(* Scaling ******************************************************************)
	IF MaxValue <> MinValue 
	THEN
		Q 													:= Offset + Scale(In , SEL(Options.0, 0.0, SEL(Options.4, -32768.0, -7629.0)), 32767.0, MinValue , MaxValue);
		IF NoOfDigits > 0
		THEN
			Q												:= TO_FMLREAL(Q,NoOfDigits);
		END_IF
	
	ELSIF NoOfDigits > 0 (* Bsp PT100 *)
	THEN
		Q													:= Offset + TO_FMLREAL(In,NoOfDigits);
		
	ELSE  													
		Q 													:= 0.0;
	END_IF

	IF 	Error AND OutOnError <> 0.000000000000000001
	THEN
		Q													:= OutOnError;
	END_IF
(**********************************************************************************************************************)

{attribute 'monitoring' := 'call'}
PROPERTY PUBLIC Error : BOOL
GET
Error					:= Status.6 OR MinValue = MaxValue AND NoOfDigits = 0;
END_GET
END_PROPERTY

{attribute 'monitoring' := 'call'}
PROPERTY PUBLIC Limit_1 : BYTE
GET
Limit_1.0					:= Status.2;
Limit_1.1					:= Status.3;
END_GET
END_PROPERTY

{attribute 'monitoring' := 'call'}
PROPERTY PUBLIC Limit_2 : BYTE
GET
Limit_2.0					:= Status.4;
Limit_2.1					:= Status.5;
END_GET
END_PROPERTY

PROPERTY PUBLIC optEnableScaleExtRangeModeNeg7629 : bool
GET
optEnableScaleExtRangeModeNeg7629 := Options.4;
END_GET
SET
Options.4 := optEnableScaleExtRangeModeNeg7629;
END_SET
END_PROPERTY

PROPERTY PUBLIC optEnableScaleSignedValue : bool
GET
optEnableScaleSignedValue := Options.0;
END_GET
SET
Options.0 := optEnableScaleSignedValue;
END_SET
END_PROPERTY

{attribute 'monitoring' := 'call'}
PROPERTY PUBLIC Overrange : BOOL
GET
Overrange					:= Status.1;
END_GET
END_PROPERTY

{attribute 'monitoring' := 'call'}
PROPERTY PUBLIC SyncError : BOOL
GET
SyncError 			:= Status.13;
END_GET
END_PROPERTY

{attribute 'monitoring' := 'call'}
PROPERTY PUBLIC TxPDOState : BOOL
GET
TxPDOState					:= Status.14; //True if not valid
END_GET
END_PROPERTY

{attribute 'monitoring' := 'call'}
PROPERTY PUBLIC TxPDOToggle : BOOL
GET
TxPDOToggle						:= Status.15;
END_GET
END_PROPERTY

{attribute 'monitoring' := 'call'}
PROPERTY PUBLIC Underrange : BOOL
GET
Underrange 					:= Status.0;
END_GET
END_PROPERTY

END_FUNCTION_BLOCK

// ---- POUs/_Miscellaneous/scale.TcPOU
//Discription:	"SCALE" scales the In-Value, which goes from InLow to InHigh, between the commited OutLow and OutHigh range.
//Used for AnalogIn/Out
FUNCTION scale : LREAL
VAR_INPUT
	In				 										: LREAL;
	InLow 													: LREAL;
	InHigh 													: LREAL;
	OutLow 													: LREAL;
	OutHigh 												: LREAL;
END_VAR
VAR
	Lim														: LREAL;
	X														: LREAL;
END_VAR

IF OutHigh <> OutLow 
THEN
	X														:= InHigh - InLow;
	IF x <> 0.0             									
	THEN       
		Lim 												:= LIMIT(InLow,In,InHigh) - InLow;             									
		X		 											:= (OutHigh - OutLow) / X;
		scale 												:= (X * Lim) + OutLow;			
	ELSE                    									
		scale												:= 0.0;
	END_IF
ELSE
	scale													:= 0.0;	
END_IF

END_FUNCTION

// ---- POUs/_Miscellaneous/Conversions/TO_FMLREAL.TcPOU
{attribute 'no_check'}
//Limits the number of decimal places in a floating point variable 
//or converts an integer number into a LREAL variable with with corresponding decimal places 
FUNCTION TO_FMLREAL : LREAL
VAR_INPUT
	 In														:	ANY_NUM;	//Input value
	 Digits													:	INT (1..32);	//number of digits to be shown
END_VAR     												
VAR         												
	 Factor													:	LREAL;
	 Value													:	LREAL;
END_VAR



IF Digits <= 0
THEN
	TO_FMLREAL												:= 0.0;	
ELSIF In.TypeClass = __SYSTEM.TYPE_CLASS.TYPE_LREAL
THEN
	Factor													:=EXPT(10,Digits);
	TO_FMLREAL												:= LINT_TO_LREAL(LREAL_TO_LINT(PLREAL_TO_LREAL(IN.pValue) * Factor)) / Factor;
ELSIF In.TypeClass = __SYSTEM.TYPE_CLASS.TYPE_REAL
THEN
	Factor													:=EXPT(10,Digits);
	TO_FMLREAL												:= LINT_TO_LREAL(LREAL_TO_LINT(PREAL_TO_REAL(IN.pValue) * Factor)) / Factor;
ELSE // Integer
	Factor													:=EXPT(10,Digits);
	CASE in.TypeClass OF		
	__SYSTEM.TYPE_CLASS.TYPE_USINT:	Value					:= TO_LREAL(PUSINT_TO_USINT(IN.pValue));								
	__SYSTEM.TYPE_CLASS.TYPE_UINT:	Value					:= TO_LREAL(PUINT_TO_UINT(IN.pValue));	
	__SYSTEM.TYPE_CLASS.TYPE_UDINT:	Value					:= TO_LREAL(PUDINT_TO_UDINT(IN.pValue));	
	__SYSTEM.TYPE_CLASS.TYPE_ULINT:	Value					:= TO_LREAL(PULINT_TO_ULINT(IN.pValue));	
	__SYSTEM.TYPE_CLASS.TYPE_SINT:	Value					:= TO_LREAL(PSINT_TO_SINT(IN.pValue));	
	__SYSTEM.TYPE_CLASS.TYPE_INT:	Value					:= TO_LREAL(PINT_TO_INT(IN.pValue));	
	__SYSTEM.TYPE_CLASS.TYPE_DINT:	Value					:= TO_LREAL(PDINT_TO_DINT(IN.pValue));	
	__SYSTEM.TYPE_CLASS.TYPE_LINT:	Value					:= TO_LREAL(PLINT_TO_LINT(IN.pValue));	
	ELSE
		TO_FMLREAL											:= 0.0;
		RETURN;
	END_CASE

	TO_FMLREAL												:= Value / Factor;
END_IF

END_FUNCTION

// ---- POUs/IO/Analog/AnalogIn32.TcPOU
{attribute 'no_check'}
FUNCTION_BLOCK AnalogIn32 extends EcSlaveInfoDataExt
VAR_INPUT
	MinValue												: 	LREAL 	:= 0.0;
	MaxValue												: 	LREAL 	:= 0.0;
	NoOfDigits												: 	INT 	(0..10)	:= 0; //number of decimal digits of scaled Q variable 
	OutOnError												:	LREAL 	:= 0.000000000000000001;
{attribute 'displaymode':='binary'}     	            	
	Options													:	BYTE  := 2#0000_0010; (* .0 = FALSE Scale value from 0 to e.g. 32767 / TRUE scale singed value e.g. -32768 <-> 32767 , see Options .1 and .2 for more scaling Options 
																						.1 = FALSE = 32 bit resolution / TRUE = value is based on 24 bit resolution e.g. -> -8388608.0 or 0.0 <-> 8388607.0 
																						.2 = Right adjust of 32/24 bit value -> value will be shifted by 8 bits (divided bv 256)   
																						.3 = TRUE = Enable extended range mode -> change scaling to +/-7812500 instead of r+/- 838860x *)
	Offset													:	LREAL := 0.0;
END_VAR                 									                                	            	
VAR_OUTPUT                              	            	
	Q														:	LREAL;	//scaled result value
	In											AT  %I* 	: 	DINT; 	//Hardware Input 
{attribute 'displaymode':='binary'}     	            	
	Status										AT  %I*		:	WORD := 2#0100_0000_0000_0000;	//Terminal status word -> can also be linked with status byte
END_VAR

(* read 32bit analog value 																				    *)
(* resolution process image			e.g.				/ 0V = 0 / 10V = 2147483647 / -10V = - 2147483647 	*)
(* or directly with NoOfDigits																	250 -> 25.0°*)
(************************************************************************************************************)
	
(* Scaling ******************************************************************)
	IF MaxValue <> MinValue 
	THEN
		IF Options.1 
		THEN //24 bit resolution
			IF NOT Options.3
			THEN
				Q 	 										:= Offset + Scale(SEL(Options.2 , In , In / 256.0 ) , SEL(Options.0, 0.0, -8388608.0), 8388607.0, MinValue , MaxValue);
			ELSE
		 		Q 	 										:= Offset + Scale(SEL(Options.2 , In , In / 256.0 ) , SEL(Options.0, 0.0, -7812500.0), 7812500.0, MinValue , MaxValue);
			END_IF
		ELSE //32 bit resolution 
			Q 	 											:= Offset + Scale(SEL(Options.2 , In , In / 256.0 ) , SEL(Options.0, 0.0, -2147483648.0), 2147483647.0, MinValue , MaxValue);		
		END_IF
		IF NoOfDigits > 0
		THEN
			Q												:= TO_FMLREAL(Q,NoOfDigits);
		END_IF
	
	ELSIF NoOfDigits > 0 (* Bsp PT100 *)
	THEN
		Q													:= Offset + TO_FMLREAL(In,NoOfDigits);
		
	ELSE  													
		Q 													:= 0.0;
	END_IF

	IF 	Error AND OutOnError <> 0.000000000000000001
	THEN
		Q													:= OutOnError;
	END_IF
(**********************************************************************************************************************)

{attribute 'monitoring' := 'call'}
PROPERTY PUBLIC Error : BOOL
GET
Error					:= Status.6 OR MinValue = MaxValue AND NoOfDigits = 0;
END_GET
END_PROPERTY

{attribute 'monitoring' := 'call'}
PROPERTY PUBLIC Limit_1 : BYTE
GET
Limit_1.0					:= Status.2;
Limit_1.1					:= Status.3;
END_GET
END_PROPERTY

{attribute 'monitoring' := 'call'}
PROPERTY PUBLIC Limit_2 : BYTE
GET
Limit_2.0					:= Status.4;
Limit_2.1					:= Status.5;
END_GET
END_PROPERTY

PROPERTY optEnable24BitResolution : BOOL //In value is provided as 32bit value instead if 24bit
GET
optEnable24BitResolution := Options.1;
END_GET
SET
Options.1 := optEnable24BitResolution;
END_SET
END_PROPERTY

PROPERTY PUBLIC optEnableScaleExtRangeMode : bool
GET
optEnableScaleExtRangeMode := Options.3;
END_GET
SET
Options.3 := optEnableScaleExtRangeMode;
END_SET
END_PROPERTY

PROPERTY PUBLIC optEnableScaleSignedValue : bool
GET
optEnableScaleSignedValue := Options.0;
END_GET
SET
Options.0 := optEnableScaleSignedValue;
END_SET
END_PROPERTY

PROPERTY PUBLIC optShiftValueBy8Bits : BOOL
GET
optShiftValueBy8Bits := Options.2;
END_GET
SET
Options.2 := optShiftValueBy8Bits;
END_SET
END_PROPERTY

{attribute 'monitoring' := 'call'}
PROPERTY PUBLIC Overrange : BOOL
GET
Overrange					:= Status.1;
END_GET
END_PROPERTY

{attribute 'monitoring' := 'call'}
PROPERTY PUBLIC SyncError : BOOL
GET
SyncError 			:= Status.13;
END_GET
END_PROPERTY

{attribute 'monitoring' := 'call'}
PROPERTY PUBLIC TxPDOState : BOOL
GET
TxPDOState					:= Status.14; //True if not valid
END_GET
END_PROPERTY

{attribute 'monitoring' := 'call'}
PROPERTY PUBLIC TxPDOToggle : BOOL
GET
TxPDOToggle						:= Status.15;
END_GET
END_PROPERTY

{attribute 'monitoring' := 'call'}
PROPERTY PUBLIC Underrange : BOOL
GET
Underrange 					:= Status.0;
END_GET
END_PROPERTY

END_FUNCTION_BLOCK

// ---- POUs/IO/Analog/AnalogOut.TcPOU
{attribute 'no_check'}
//Provides an INT output varibale (Q	AT  %Q* : 	INT) to writed a scaled lreal value to an anallog output (terminal)
FUNCTION_BLOCK AnalogOut
VAR_INPUT
	SetValue												: 	LREAL 	:= 0.0;	
	MinValue												: 	LREAL 	:= 0.0;
	MaxValue												: 	LREAL 	:= 0.0;	
{attribute 'displaymode':='binary'}
	Options													:	BYTE 	:= 2#0000_0000; (* .0 = FALSE scale output to 0 - 32767 / TRUE = scale output from -32768 to +32767 *)
END_VAR             							
VAR_OUTPUT          							
	Q												AT  %Q* : 	INT; (* Hardware Output *)
END_VAR             							
VAR                 							
	x														:	LREAL;
END_VAR

(* Analogvalue output	 													    *)
(* resolution  							/ 0V = 0 / 10V = 32768 / -10V = - 32767 *)
(********************************************************************************)

(* standardization **************************************************************)
	Q															:= TO_INT(Scale(SetValue,MinValue,MAxValue,SEL(Options.0 , 0.0  , -32768.0), 32767.0));		

(*********************************************************************************)

PROPERTY PUBLIC optEnableScaleSignedValue : bool
GET
optEnableScaleSignedValue := Options.0;
END_GET
SET
Options.0 := optEnableScaleSignedValue;
END_SET
END_PROPERTY

END_FUNCTION_BLOCK

// ---- POUs/IO/ButtonExt.TcPOU
{attribute 'no_check'}
//Button with delay function 
FUNCTION_BLOCK ButtonExt EXTENDS Button
VAR_INPUT
	RstTGL													:	BOOL := FALSE; 	//resets the Toggle signal
	SetTGL													:	BOOL := FALSE;	//sets the Toggle signal

	PT_ON													:	TIME := T#0MS; 	//Delay for Q, Q_RT (TGL) and Q_FT
END_VAR
VAR_OUTPUT
	Q_DIRECT												:	BOOL; 	//Direct signal - undelayed
END_VAR
VAR
	TON														:	TON;
END_VAR

(* Button with toggle-function and on-delay		V1.5	*)
(********************************************************)

(********************************************************)
TON(IN := ((In OR Force) XOR Invert) AND Enable, PT := PT_ON);
Q_DIRECT 													:= TON.IN;
IF NOT Q    												
THEN        												
	Q 														:= TON.Q;
	Q_RT 													:= Q;
	Q_FT 													:= FALSE;
ELSE        												
	Q 														:= TON.IN;
	Q_RT 													:= FALSE;
	Q_FT 													:= NOT Q;
END_IF      	

Q_TGL := NOT RstTGL AND (Q_RT XOR Q_TGL OR SetTGL) ;

(********************************************************)

END_FUNCTION_BLOCK

// ---- POUs/IO/Drives/Stepper/AxDriveStepper_wEvents.TcPOU
{attribute 'no_check'}
//Beckhoff Stepper terminal diag and diagnosis with eventlogger - extended from AxDriveStepper
//EventHandling instance use inside
FUNCTION_BLOCK AxDriveStepper_wEvents EXTENDS AxDriveStepper
VAR CONSTANT         	
END_VAR  
VAR_INPUT
	EnableEvent												:	BOOL := TRUE; //Enable to show events
	ConfirmTrig												:	BOOL := FALSE; //Quit events
	SourceId												:	UDINT := 102600; //MDP742 Stepper CoE Drive default multisource Id + Ax id
	Name													:	STRING(30) := '';
	ErrorLimitPos											:	BOOL := FALSE;
	ErrorLimitNeg											:	BOOL := FALSE;
END_VAR                     					
VAR_IN_OUT                  					
END_VAR                     					
VAR_OUTPUT                  					
 	EventStatus												:	DWORD;       
	NoOfActiveEvents										:	INT;                    					
END_VAR                     					                   					
VAR                         					
END_VAR
VAR

(* Cache *********************************************************************)
	
(* Timer ********************************************************************************)

(* Trigger ******************************************************************************)

(* Instance ****************************************************************************)
	Event													:	EventHandlingGrp10;
	
(* Dummy Speicher **********************************************************)
	i														: INT := 0 ;
END_VAR

	(* Stepper Drive Control with events												*)
	(************************************************************************************)

(* Call super **********************************************)
	SUPER^();
	
(* work events *******************************************)
	_callEvents();

(*******************************************************)

METHOD PRIVATE _callEvents : BOOL
VAR_INPUT
END_VAR

(* Check if msg activ and init some parameter ***********************)
	IF Event.no[1].Text2 <> Name AND Name <> '' OR Event.no[1].Text2 = '' AND rAxis.NcToPlc.AxisId <> 0
	THEN
		Event.no[1].eClass 									:= TC2_SYSTEM.TCEVENTCLASS_STATEINFO;
		Event.no[3].eClass 									:= TC2_SYSTEM.TCEVENTCLASS_MESSAGE;
		
		(* Init Achsname *)
		FOR i := Event.MIN_EVENT TO Event.MAX_EVENT DO
		(*	Event.no[i].Text1								:= '';*)
			Event.no[i].Text2								:= SEL(LEN(name)>1,CONCAT('Axis id:',DWORD_TO_STRING(rAxis.NcToPlc.AxisId)),name);
		END_FOR
	END_IF

(* workl Event Ctrl *************************************************)
	Event(
		ConfirmTrig := ConfirmTrig,
		Disable		:= rAxis.NcToPlc.AxisId = 0 OR NOT EnableEvent,
		SourceId	:= SourceId + rAxis.NcToPlc.AxisId,
		Status		=> EventStatus,
		NoOfActiveEvents => NoOfActiveEvents);

(* Event Logger Meldungen *****************************************************)
	Event.no[1].Flag 										:= NOT Status_ReadyToEnable ; 
	Event.no[2].Flag 										:= Fault;
	Event.no[3].Flag 										:= (Status_Warning OR Diag_Configuration) AND NOT rAxis.Status.Homing AND rAxis.Status.Operational; //Avoid warning if drive is disabled (EL7037 and older FW on EL7047 <=06 - 2020-03-26) 				
	Event.no[4].Flag 										:= Diag_TorqueOverloaded;
	Event.no[5].Flag 										:= Diag_UnderVoltage OR Diag_OverVoltage OR Diag_NoControlPower;
	Event.no[6].Flag 										:= Diag_ShortCircuit OR Diag_ShortCircuitB OR Diag_OpenLoadA OR Diag_OpenLoadB; 
	Event.no[7].Flag 										:= Diag_Saturated;
	Event.no[8].Flag										:= Diag_OverTemperature ;
	Event.no[9].Flag 										:= ErrorLimitPos; 	
	Event.no[10].Flag 										:= ErrorLimitNeg;	
(*	Event.no[11].Flag 										:= FALSE; 				
	Event.no[12].Flag 										:= FALSE;					
	Event.no[13].Flag 										:= FALSE; 			Event.no[9].Class := TC2_SYSTEM.TCEVENTCLASS_WARNING;
	Event.no[14].Flag 										:= FALSE; 			Event.no[10].Class := TC2_SYSTEM.TCEVENTCLASS_WARNING;
	Event.no[15].Flag 										:= FALSE;
	Event.no[16].Flag 										:= FALSE;
	Event.no[17].Flag 										:= FALSE;
	Event.no[18].Flag 										:= FALSE;
	Event.no[19].Flag 										:= FALSE;
	Event.no[20].Flag 										:= FALSE;
	Event.no[21].Flag 										:= FALSE;
	Event.no[22].Flag 										:= FALSE;
	Event.no[23].Flag 										:= FALSE;
	Event.no[24].Flag 										:= FALSE;
	Event.no[25].Flag 										:= FALSE;
*)

(******************************************************************************)
END_METHOD

METHOD PUBLIC confirm : bool
VAR_INPUT
END_VAR
confirm			:= Event.confirm();
END_METHOD

END_FUNCTION_BLOCK

// ---- POUs/IO/EL-EP/AnalogOut_EL2535.TcPOU
{attribute 'no_check'}
FUNCTION_BLOCK AnalogOut_EL2535 EXTENDS AnalogOut
VAR_INPUT
	Reset										AT  %Q*		:	BOOL;	
END_VAR   
VAR_IN_OUT
END_VAR              									                              	            	
VAR_OUTPUT                              	            	
	Input										AT  %I* 	: 	BOOL; 	//Hardware Input 
	ReadyToEnable								AT  %I* 	: 	BOOL; 	
	Warning										AT  %I* 	: 	BOOL; 	
	Error										AT  %I* 	: 	BOOL; 	
	TxPDOToggle									AT  %I* 	: 	BOOL; 	
            
	InfoData1									AT  %I* 	: 	INT; //Actual current
	InfoData2									AT  %I* 	: 	INT; //Duty cycle/Voltage
END_VAR                                 	
VAR                                     	
END_VAR

(* Set PWM Output of EL25xx																					*)
(************************************************************************************************************)
	SUPER^();

(********************************************************************************************************)

END_FUNCTION_BLOCK

// ---- POUs/IO/EL-EP/EL3681.TcPOU
FUNCTION_BLOCK EL3681 EXTENDS EcSlaveInfoDataExt
VAR_INPUT
	MinValue												: 	LREAL 	:= 0.0;
	MaxValue												: 	LREAL 	:= 0.0;
	NoOfDigits												: 	INT 	(0..10)	:= 6; //number of decimal digits of scaled Q variable 
	OutOnError												:	LREAL 	:= 0.000000000000000001;
{attribute 'displaymode':='binary'}     	            	
	Options													:	BYTE  := 2#0000_0010; (* .0 = FALSE Scale value from 0 to e.g. 32767 / TRUE scale singed value e.g. -32768 <-> 32767 , see Options .1 and .2 for more scaling Options 
																						.1 = FALSE = 32 bit resolution / TRUE = value is based on 24 bit resolution e.g. -> -8388608.0 or 0.0 <-> 8388607.0 
																						.2 = Right adjust of 32/24 bit value -> value will be shifted by 8 bits (divided bv 256)   
																						.3 = TRUE = Enable extended range mode -> change scaling to +/-7812500 instead of r+/- 838860x *)
	Offset													:	LREAL := 0.0;
END_VAR                 									                                	            	
VAR_OUTPUT                              	            	
	Q														:	LREAL;	//scaled result value
{attribute 'displaymode':='binary'}     	            	
	Status										AT  %I*		:	WORD := 2#0100_0000_0000_0000;	//Terminal status word -> can also be linked with status byte

	In											AT  %I* 	: 	DINT; 	//Hardware Input 

	ActMode													: 	BYTE; //Setting Mode: 	0 = [V] DC | 1 = [V] AC 	| 2 = [A] DC 	| 3 = [A] AC
	ActRange												: 	BYTE; //Setting Range: 255 = 0.3 	| 1 = 3 		| 2 = 30 		| 3 = 300 

{attribute 'displaymode':='hex'}
	Control										AT%Q*		: 	WORD;   
    	
END_VAR
VAR	
{attribute 'displaymode':='hex'}
	Settings									AT  %I*		:	WORD; //Actual setting for mode and range 
END_VAR

SUPER^();

(* Scaling ******************************************************************)
	IF MaxValue <> MinValue 
	THEN
		IF Options.1 
		THEN //24 bit resolution
			IF NOT Options.3
			THEN
				Q 	 										:= Offset + Scale(SEL(Options.2 , In , In / 256.0 ) , SEL(Options.0, 0.0, -8388608.0), 8388607.0, MinValue , MaxValue);
			ELSE
		 		Q 	 										:= Offset + Scale(SEL(Options.2 , In , In / 256.0 ) , SEL(Options.0, 0.0, -7812500.0), 7812500.0, MinValue , MaxValue);
			END_IF
		ELSE //32 bit resolution 
			Q 	 											:= Offset + Scale(SEL(Options.2 , In , In / 256.0 ) , SEL(Options.0, 0.0, -2147483648.0), 2147483647.0, MinValue , MaxValue);		
		END_IF
		IF NoOfDigits > 0
		THEN
			Q												:= TO_FMLREAL(Q,NoOfDigits);
		END_IF
	
	ELSIF NoOfDigits > 0 (* Bsp PT100 *)
	THEN
		Q													:= Offset + TO_FMLREAL(In,NoOfDigits);
		
	ELSE  													
		Q 													:= 0.0;
	END_IF

	IF inError AND OutOnError <> 0.000000000000000001
	THEN
		Q													:= OutOnError;
	END_IF
	
(* Mode & Range **************************************************************)
	ActMode.0 												:= Settings.4;
	ActMode.1 												:= Settings.5;
	ActMode.2 												:= Settings.6;
	ActMode.3 												:= Settings.7;
	
	ActRange.0 												:= Settings.8;
	ActRange.1 												:= Settings.9;
	ActRange.2 												:= Settings.10;
	ActRange.3 												:= Settings.11;
	ActRange.4 												:= Settings.12;
    ActRange.5 												:= Settings.13;
    ActRange.6 												:= Settings.14;
    ActRange.7 												:= Settings.15;

(*****************************************************************************)

{attribute 'monitoring' := 'call'}
PROPERTY PUBLIC autorangeIsDisabled : BOOL
GET
autorangeIsDisabled := Status.5;
END_GET
END_PROPERTY

{attribute 'monitoring' := 'call'}
PROPERTY PUBLIC calibrationInProgress : BOOL
GET
calibrationInProgress := Status.7;
END_GET
END_PROPERTY

{attribute 'monitoring' := 'call'}
PROPERTY PUBLIC dataInvalid : BOOL
GET
dataInvalid := Status.3;
END_GET
END_PROPERTY

{attribute 'monitoring' := 'call'}
PROPERTY PUBLIC disableAutorange : BOOL
GET
DisableAutorange 	:= Control.0;
END_GET
SET
Control.0 								:= DisableAutorange;
END_SET
END_PROPERTY

{attribute 'monitoring' := 'call'}
PROPERTY PUBLIC inError : BOOL
GET
InError					:= Status.6 OR MinValue = MaxValue AND NoOfDigits = 0;
END_GET
END_PROPERTY

{attribute 'monitoring' := 'call'}
PROPERTY PUBLIC inExtendedRange : BOOL
GET
inExtendedRange := Status.2;
END_GET
END_PROPERTY

{attribute 'monitoring' := 'call'}
PROPERTY PUBLIC overrange : BOOL
GET
overrange 		:= status.1;
END_GET
END_PROPERTY

{attribute 'monitoring' := 'call'}
PROPERTY PUBLIC rangeInvalid : BOOL
GET
rangeInvalid := Status.4;
END_GET
END_PROPERTY

{attribute 'monitoring' := 'call'}
// 0 = [V] DC | 1 = [V] AC | 2 = [A] DC | 3 = [A] AC
PROPERTY PUBLIC setControlMode : INT
GET
setControlMode.0 := Control.4;
setControlMode.1 := Control.5;
setControlMode.2 := Control.6;
setControlMode.3 := Control.7;
END_GET
SET
Control.4 := setControlMode.0;
Control.5 := setControlMode.1;
Control.6 := setControlMode.2;
Control.7 := setControlMode.3;
END_SET
END_PROPERTY

{attribute 'monitoring' := 'call'}
// 	disable autorange to use range
// 	255 = 0.3 		| 1 = 3 		| 2 = 30 		| 3 = 300 
//	255 = 3*10^-1 	| 1 = 3*10^0 	| 2 = 3*10^1 	| 3 = 3*10^2 
PROPERTY PUBLIC setControlRange : INT
GET
setControlRange.0 := Control.8;
setControlRange.1 := Control.9;
setControlRange.2 := Control.10;
setControlRange.3 := Control.11;
setControlRange.4 := Control.12;
setControlRange.5 := Control.13;
setControlRange.6 := Control.14;
setControlRange.7 := Control.15;
END_GET
SET
Control.8 := setControlRange.0;
Control.9 := setControlRange.1;
Control.10 := setControlRange.2;
Control.11 := setControlRange.3;
Control.12 := setControlRange.4;
Control.13 := setControlRange.5;
Control.14 := setControlRange.6;
Control.15 := setControlRange.7;
END_SET
END_PROPERTY

{attribute 'monitoring' := 'call'}
PROPERTY PUBLIC startCalibration : BOOL
GET
StartCalibration 	:= Control.1;
END_GET
SET
Control.1 								:= StartCalibration;
END_SET
END_PROPERTY

{attribute 'monitoring' := 'call'}
PROPERTY PUBLIC underrange : BOOL
GET
underrange 		:= status.0;
END_GET
END_PROPERTY

END_FUNCTION_BLOCK

// ---- POUs/IO/_EcSlaveFWUpdater/EcSlaveDevFWUpdater.TcPOU
FUNCTION_BLOCK EcSlaveDevFWUpdater EXTENDS FbBase
VAR CONSTANT	
	{attribute 'displaymode':='hexadecimal'} 
	COE_FWVERSION_OBJECT								: WORD := 16#100A;
END_VAR
VAR_OUTPUT CONSTANT
	MIN_SLAVE_DEV										:	INT := 1;
	MAX_SLAVE_DEV										:	INT := Param.ETHERCAT_SLAVE_DEV_FW_UPDATER_MAX_DEV;

	{attribute 'displaymode':='binary'}   
	MODE_READ											:	BYTE := 0;
	{attribute 'displaymode':='binary'}   
	MODE_WRITE											:	BYTE := 1;

	{attribute 'displaymode':='binary'}   
	OPTION_WRITE_FW_IF_VERSION_MATCH					:	BYTE := 2#0000_0001;
	
END_VAR
VAR_INPUT
{attribute 'displaymode':='binary'}         			
	Mode												:	BYTE  := 2#0000_0000; 

{attribute 'displaymode':='binary'}  	
	Options												:	BYTE  := 2#0000_0000; 		
				
	PathName											:	STRING; //Path incl. file name of FW file
	RegVersion											:	STRING; //Requested version
	ipSlaveInfoData										:	ARRAY [MIN_SLAVE_DEV..MAX_SLAVE_DEV] OF I_EcSlaveInfoData;
END_VAR
VAR_OUTPUT
	ActVersion											: ARRAY[MIN_SLAVE_DEV..MAX_SLAVE_DEV] OF STRING[20]; 	
	CntFWNOK											: INT; //Count of terminals FW not OK
	TermNo												: INT; //No of terminal in progress
	ProgressWriteFW										: UDINT;	
	VersionRead											: BOOL;
END_VAR
VAR
(*  Memory *****************************************************)
	lastState											: INT := 0;
	MinTerm												: INT;

(*  Timer ******************************************************)
(*  Trigger ****************************************************)

(*  Blocks *****************************************************)
	EcCoeSdoReadEx										: FB_EcCoeSdoReadEx := (nIndex := COE_FWVERSION_OBJECT, tTimeout := DEFAULT_ADS_TIMEOUT);

	CoEFwDownLoad										: FB_EcFoeLoad := (tTimeout := DEFAULT_ADS_TIMEOUT,dwPass := 0, eMode := eFoeMode_Write);
(*  Error ******************************************************)
(*  Dummys *****************************************************)
	{attribute 'hide' := ''}
	i,j													: INT := 0;

END_VAR

	(*********************************************************)
	
(* state machine ********************************************************)
	rtExecute(CLK := Execute);
	CASE state OF
	0 : 
		Busy 											:= FALSE;
		
		IF NOT Execute THEN
			Done 										:= FALSE;
			Error 										:= FALSE;
			ErrorID 									:= 0;
		END_IF
		IF rtExecute.Q THEN
			IF PathName = '' 
			THEN
				Error 									:= TRUE;
				ErrorID 								:= E_AdsErr.DEVICE_INVALIDPARM;

			ELSIF RegVersion = '' AND Mode = MODE_WRITE AND NOT Options.0
			THEN
 				Error 									:= TRUE;
				ErrorID 								:= E_AdsErr.DEVICE_INVALIDPARM; 
									
			ELSIF ipSlaveInfoData[MIN_SLAVE_DEV] = 0
			THEN
 				Error 									:= TRUE;
				ErrorID 								:= E_AdsErr.DEVICE_INVALIDPARM; 			
			ELSE
				Busy									:= TRUE;	
				Done 									:= FALSE;
				Error 									:= FALSE;
				ErrorID 								:= 0;
				TermNo									:= MIN_SLAVE_DEV;	
				ProgressWriteFW							:= 0;
				CntFWNOK								:= 0;					
				
			
				EcCoeSdoReadEx(bExecute := FALSE);
				CoEFwDownLoad(bExecute := FALSE);
				state									:= SEL(Mode = MODE_READ, 1, 2);
			END_IF
		END_IF
			
	1: (* Write FW *****************************************************************)
		CoEFwDownLoad(
			bExecute		:= ipSlaveInfoData[TermNo].rInfoData.AdsAddr.port <> 0 AND (ActVersion[TermNo] <> RegVersion OR Options.0) , 
			sNetId			:= F_CreateAmsNetId(nIds := ipSlaveInfoData[TermNo].rInfoData.AdsAddr.netId),
			nSlaveAddr		:= ipSlaveInfoData[TermNo].rInfoData.AdsAddr.port,
			sPathName		:= PathName,
			nProgress 		=> ProgressWriteFW);	
		IF NOT 	CoEFwDownLoad.bBusy
		THEN
			ProgressWriteFW								:= 0;
			IF CoEFwDownLoad.bError
			THEN
				ErrorID									:= EcCoESdoReadEx.nErrId;
				CntFWNOK								:= CntFWNOK + 1;	
				ActVersion[TermNo]						:= 'ERR_DOWNLOADING';
			ELSIF CoEFwDownLoad.bExecute	
			THEN
				ActVersion[TermNo]						:= 'DOWNLOADED';
			ELSE
				ActVersion[TermNo]						:= '------';
			END_IF
			//Next terminal
			TermNo										:= TermNo + 1;
			
			IF TermNo > MAX_SLAVE_DEV 
				OR ipSlaveInfoData[TermNo] = 0
			THEN //Start reading
				MEMSET(ADR(ActVersion),0,SIZEOF(ActVersion));
				VersionRead								:= FALSE;
				TermNo									:= MIN_SLAVE_DEV;		
				state									:= 2;
			END_IF		
			CoEFwDownLoad(bExecute := FALSE);
		ELSE
			ActVersion[TermNo]							:= CONCAT('DOWNLOADING ',CONCAT(TO_STRING(CoEFwDownLoad.nProgress),'%'));
		END_IF
	
	2: (* Read FW Version **********************************************************)
		EcCoESdoReadEx(
			bExecute		:= ipSlaveInfoData[TermNo].rInfoData.AdsAddr.port <> 0,
			sNetId			:= F_CreateAmsNetId(nIds := ipSlaveInfoData[TermNo].rInfoData.AdsAddr.netId),
			nSlaveAddr		:= ipSlaveInfoData[TermNo].rInfoData.AdsAddr.port,
			pDstBuf			:= ADR(ActVersion[TermNo]),
			cbBufLen		:= SIZEOF(ActVersion[TermNo]));
		IF NOT EcCoESdoReadEx.bBusy
		THEN
			IF EcCoESdoReadEx.bError 
			THEN
				ActVersion[TermNo]						:= 'ERR_READING';
				ErrorID									:= EcCoESdoReadEx.nErrId;
				CntFWNOK								:= CntFWNOK + 1;	
			ELSIF NOT EcCoESdoReadEx.bExecute 
			THEN
				ActVersion[TermNo]						:= 'NOT_CONNECTED';
			ELSIF ActVersion[TermNo] <> RegVersion
			THEN
				CntFWNOK								:= CntFWNOK + 1;	
			END_IF
			
			//Next terminal
			TermNo										:= TermNo + 1;
			
			IF TermNo > MAX_SLAVE_DEV
				OR ipSlaveInfoData[TermNo] = 0
			THEN
				TermNo									:= MAX_SLAVE_DEV;
				Done									:= CntFWNOK = 0;
				VersionRead								:= TRUE;
				Error									:= NOT Done;
				Busy									:= FALSE;
				state									:= 0;
			END_IF
			EcCoeSdoReadEx(bExecute := FALSE);
		END_IF
	END_CASE	

(* Record last state ******************************************)
IF state <> lastState AND state <> 0 AND NOT Error
THEN 
	lastState											:= state;
END_IF

(*************************************************************)

END_FUNCTION_BLOCK

// ---- POUs/IO/_EcSlaveInfoDataIO/EcSlaveInfoData.TcPOU
{attribute 'no_check'}
FUNCTION_BLOCK EcSlaveInfoData implements I_EcSlaveInfoData
VAR_INPUT
END_VAR
VAR_OUTPUT
	WcState											AT  %I*		:	BOOL;			//TRUE=Invalid - TRUE an invalid working counter and FALSE a valid working counter 
	InputToggle										AT  %I*		:	BOOL;			//variable toggles in every successful cycle	
	{attribute 'displaymode':='hex'}  
	InfoDataState									AT  %I*		: 	UINT;			(* current EtherCAT device state:
																						EC_DEVICE_STATE_MASK		:BYTE 	:=16#0F;
																						EC_DEVICE_STATE_INIT		:BYTE 	:=16#01;
																						EC_DEVICE_STATE_PREOP		:BYTE 	:=16#02;
																						EC_DEVICE_STATE_BOOTSTRAP	:BYTE 	:=16#03;
																						EC_DEVICE_STATE_SAFEOP		:BYTE 	:=16#04;
																						EC_DEVICE_STATE_OP			:BYTE 	:=16#08;
																						EC_DEVICE_STATE_ERROR		:BYTE 	:=16#10;
																						EC_DEVICE_STATE_INVALID_VPRS :BYTE 	:=16#20;
																						EC_DEVICE_STATE_INITCMD_ERROR:BYTE 	:=16#40; *)
	AdsAddr											AT  %I*		:	AMSADDR; 		//Slave device AdsAddr structure(ID and port number)
END_VAR
VAR
END_VAR

;

PROPERTY PUBLIC rInfoData : reference to EcSlaveInfoData
GET
rInfoData := THis^;
END_GET
END_PROPERTY

END_FUNCTION_BLOCK

// ---- POUs/IO/EL-EP/EL1904.TcPOU
{attribute 'no_check'}
FUNCTION_BLOCK EL1904 (* EL Safety Input Terminal IO *)
VAR_INPUT
END_VAR
VAR_OUTPUT
	C1												AT  %I* : BOOL;	//TRUE when channel 1 has high signal
	C2												AT  %I* : BOOL;	//TRUE when channel 2 has high signal
	C3												AT  %I* : BOOL;	//TRUE when channel 3 has high signal
	C4												AT  %I* : BOOL;	//TRUE when channel 4 has high signal
	Valid													: BOOL;	//TRUE when data is valid
END_VAR		            							
VAR                     							
	FSoESlaveCMD									AT  %I* : USINT;
END_VAR

(* EL 1904 Terminal Inputs					             	 V1.2	*)
(********************************************************************)

(* Input Signals Valid ******************************************************)
	Valid 													:= FSoESlaveCMD = 16#36
																	OR FSoESlaveCMD = 16#08;
          													
(**********************************************************************)

END_FUNCTION_BLOCK

// ---- POUs/IO/EL-EP/EL3403/EL3403.TcPOU
{attribute 'no_check'}
FUNCTION_BLOCK EL3403 Extends EcSlaveInfoData
VAR CONSTANT
	MIN_PHASE												:	INT := 1;
	MAX_PHASE												:	INT := 3;
END_VAR  
VAR_INPUT
	IndexOut										AT %Q*	:	ARRAY[MIN_PHASE..MAX_PHASE] OF USINT;
	Transmission											:	ARRAY[MIN_PHASE..MAX_PHASE] OF LREAL;	//Transmission current transformator for each phase e.g. 750 *)
END_VAR
VAR_OUTPUT
	(* Inputs Channel 1-3 *)
	TxPDOToggle										AT %I*	: 	ARRAY[MIN_PHASE..MAX_PHASE] OF BOOL;
	IndexIn											AT %I*	: 	ARRAY[MIN_PHASE..MAX_PHASE] OF USINT;
	Current													: 	ARRAY[MIN_PHASE..MAX_PHASE] OF LREAL; 	//Unit: 0,000001 A
	Voltage													: 	ARRAY[MIN_PHASE..MAX_PHASE] OF LREAL; 	//Unit: 0,0001 V
	ActivePower												: 	ARRAY[MIN_PHASE..MAX_PHASE] OF LREAL; 	//Unit: 0,01 W

	(* PM Status Data *)
	MissingZeroCrossingA							AT %I*	: 	BOOL;
	MissingZeroCrossingB							AT %I* 	: 	BOOL;
	MissingZeroCrossingC							AT %I* 	: 	BOOL;
	PhaseSequenceError								AT %I* 	: 	BOOL;
//	SyncError										AT %I* 	: 	BOOL;
                                                              	
	(* MultiplexValues	*)
	ApparentPower											:	ARRAY[MIN_PHASE..MAX_PHASE] OF LREAL; 	//apparent power unit: 0,01 VA
	ReactivePower											:	ARRAY[MIN_PHASE..MAX_PHASE] OF LREAL; 	//reactive power unit: 0,01 VAr
	PowerFactor												:	ARRAY[MIN_PHASE..MAX_PHASE] OF LREAL; 	//effective power cos phi Unit: 0,001
	EnergyConsumption										:	ARRAY[MIN_PHASE..MAX_PHASE] OF LREAL; 	//energy unit: 0,001 Wh
	EnergyConsumptionInvers									:	ARRAY[MIN_PHASE..MAX_PHASE] OF LREAL; 	//energy unit: 0,001 Wh
	TimestampDistClocks										:	ARRAY[MIN_PHASE..MAX_PHASE] OF LREAL; 	//timestamp unit : 1 ns
	Frequency												:	ARRAY[MIN_PHASE..MAX_PHASE] OF LREAL; 	//frequenzy unit : 0,1 Hz

END_VAR
VAR (* Internal IOs *)
	_Current										AT %I* 	: 	ARRAY[MIN_PHASE..MAX_PHASE] OF DINT; 	//Unit: 0,000001 A
	_Voltage										AT %I* 	: 	ARRAY[MIN_PHASE..MAX_PHASE] OF DINT; 	//Unit: 0,0001 V
	_ActivePower									AT %I* 	: 	ARRAY[MIN_PHASE..MAX_PHASE] OF DINT; 	//Unit: 0,01 W

	_VariantValue									AT %I* 	: 	ARRAY[MIN_PHASE..MAX_PHASE] OF DINT;
//	_SyncErrorChannel								AT %I* 	: 	ARRAY[MIN_PHASE..MAX_PHASE] OF BOOL; 	//reserved
//	_SyncErrorTerminal										: 	BOOL;	//reserved
END_VAR                       							
VAR
	i														:	INT;
END_VAR

(* EL 3403 IO 									*)
(************************************************)

(* Get Index Values *****************************)
	FOR i := MIN_PHASE TO MAX_PHASE DO
		Current[i]											:= Transmission[i] * DINT_TO_LREAL(_Current[i]) / 1000000.0; //A
		Voltage[i]											:= (*Uebersetzung[i] **) DINT_TO_LREAL(_Voltage[i]) / 10000.0; //V
		ActivePower[i]										:= Transmission[i] * DINT_TO_LREAL(_ActivePower[i]) / 100.0; //W
                                            				
		CASE IndexIn[i] OF                  				
		0:(*Scheinleistung*)                				
			ApparentPower[i]								:= Transmission[i] * DINT_TO_LREAL(_VariantValue[i]) / 100.0; //VA
                                            				
		1:(*Blindleistung*)                 				
			ReactivePower[i]								:= Transmission[i] * DINT_TO_LREAL(_VariantValue[i]) / 100.0; //VAr
                                            				
		2:(*Energie*)                       				
			EnergyConsumption[i]							:= Transmission[i] * DINT_TO_LREAL(_VariantValue[i]) / 1000.0; //Wh
                                            				
		3:(*Wirkleistungsfaktor*)           				
			PowerFactor[i]									:= DINT_TO_LREAL(_VariantValue[i]) / 1000.0; //cos phi
                                            				
		4:(*Frequenz*)                      	
			Frequency[i]									:= DINT_TO_LREAL(_VariantValue[i]) / 10.0; //Hz
                                            				
		5:(*Energie Invers*)                				
			EnergyConsumptionInvers[i]						:= Transmission[i] * DINT_TO_LREAL(_VariantValue[i]) / 1000.0;
                                            				
		100:(*Zeitstempel*)                 				
			TimestampDistClocks[i]							:= DINT_TO_LREAL(_VariantValue[i]);
	
		END_CASE

	END_FOR

(***********************************************)

END_FUNCTION_BLOCK

// ---- POUs/IO/InOutExt.TcPOU
{attribute 'no_check'}
FUNCTION_BLOCK InOutExt EXTENDS InOut IMPLEMENTS I_ActuatorOnOff
VAR_INPUT
	ResetTrig												:	BOOL;	//Resets error with rising edge
	Invert													:	BOOL ;			//Inverts the logic of varibale In (AT  %I*)
	PT_Timeout												:	TIME := T#3S;  	//Time value until Timeout of process (Error)
END_VAR                     				
VAR_OUTPUT                  				
	Busy													:	BOOL;			//Busy is TRUE at the rising edge of Execute and FALSE when one of the outputs Done, Aborted, or Error is set 
	ErrorOn													:	BOOL;			//Timeout error waiting for IN changing to TRUE
	ErrorOff												:	BOOL;			//Timeout error waiting for IN changing to FALSE
	Done													:	BOOL;			//The Done output is set when the commanded action has been completed successfully 
	Status													:	BYTE;			//8 different query Options (conditions see below)
END_VAR                     	
VAR                         	
	tonRM													:	ton;			
END_VAR

(* Actuator with feedback								*)
(********************************************************)

(********************************************************)
	IF Q 
	THEN
		SwitchOn();
	ELSE
		SwitchOff();
	END_IF
	_runtimeChk();
	_writeStatus();

(********************************************************)

METHOD PROTECTED _runtimeChk : BOOL
VAR_INPUT
END_VAR
	tonRM(
		IN	:= Busy AND NOT ResetTrig,  
		PT 	:= PT_Timeout,
		Q	=> );
		
	ErrorOff 												:= tonRM.Q AND NOT Q;
	ErrorOn 												:= tonRM.Q AND Q;

	_runtimeChk									:= TRUE;
END_METHOD

METHOD PROTECTED _writeStatus : BOOL
VAR_INPUT
END_VAR
	Status.0 												:= NOT Q;
	Status.1 												:= Q;
	Status.2 												:= NOT (In XOR Invert);
	Status.3 												:= In XOR Invert;
	Status.4 												:= NOT ErrorOff;
	Status.5 												:= NOT ErrorOn;
	Status.6 												:= NOT Status.7;
	Status.7 												:= ErrorOff OR ErrorOn;
	
	(* Result *)
	_writeStatus											:= TRUE;
END_METHOD

METHOD PUBLIC enable : BOOL //Result value = TRUE if successful executed (
VAR_INPUT 
	IN								: BOOL; //TRUE = ON/FALSE = OFF	
END_VAR
IF IN
THEN
	enable							:= switchOn();
ELSE
	enable							:= switchOff();
END_IF
END_METHOD

{attribute 'monitoring' := 'call'}
PROPERTY public inError : BOOL
GET
inError := ErrorON or ErrorOff;
END_GET
END_PROPERTY

{attribute 'monitoring' := 'call'}
PROPERTY public isBusy : bool
GET
isBusy := Busy;
END_GET
END_PROPERTY

{attribute 'monitoring' := 'call'}
PROPERTY public isOff : BOOL
GET
isOff := not Q;
END_GET
END_PROPERTY

{attribute 'monitoring' := 'call'}
PROPERTY public isOn : BOOL
GET
isOn := Q;
END_GET
END_PROPERTY

{attribute 'monitoring' := 'call'}
PROPERTY Public noFeed : BOOL
GET
noFeed := FALSE;
END_GET
END_PROPERTY

{attribute 'monitoring' := 'call'}
PROPERTY Public ok : bool
GET
ok := Q and Done or not Q and not Done;
END_GET
END_PROPERTY

METHOD PUBLIC reset : Bool
VAR_INPUT
END_VAR
tonRM(IN := FALSE);
reset := TRUE;
END_METHOD

METHOD public switchOff : BOOL
VAR_INPUT
END_VAR
	
	Q														:= FALSE;
	Done													:= NOT (In XOR Invert);
	Busy													:= NOT Done;
	switchOff												:= Done;
END_METHOD

METHOD public switchOn : BOOL
VAR_INPUT
END_VAR
	Q														:= TRUE;
	Done													:= (In XOR Invert);
	Busy													:= NOT Done;
	switchOn												:= Done;
END_METHOD

END_FUNCTION_BLOCK

// ---- POUs/IO/Motors/IOMotor2Dir.TcPOU
{attribute 'no_check'}
FUNCTION_BLOCK IOMotor2Dir EXTENDS IOMotor IMPLEMENTS I_ActuatorFwdRev
VAR_INPUT
	StartBwd													:	BOOL; 
	FeedBwd														:	BOOL := TRUE;
END_VAR                 					
VAR_OUTPUT              					
	Q_ContactorBwd									AT  %Q* 	:	BOOL; //Hardware output for contactor to move backwards
END_VAR                 					
VAR 					
END_VAR                 	
VAR                     	
END_VAR

(* Com Motor IO 2 Directions		 		V2.2 	*)
(****************************************************)

(* Protection Switch *****************************************)
	IF ResetTrig 
	THEN 
		reset(); 
	END_IF
	
	ProtSwitchOK();
	
(* Enable ****************************************************)
	IF 	Start 
		AND NOT StartBwd 
	THEN
		startForward();
	ELSIF StartBwd 
		AND NOT Start 
	THEN
		startReverse();
	ELSE
		switchOff();
	END_IF
	
(* HMI status *********************************************)
	_writeStatus();
	
(********************************************************)

METHOD PROTECTED _writeStatus : BOOL
VAR_INPUT
END_VAR
	
(* HmiStatus **************************************************)
	Status.0 												:= Q_Contactor;
	Status.1 												:= Q_ContactorBwd;
	Status.2 												:= FALSE;
	Status.3 												:= FALSE;
	Status.4 												:= Feed;
	Status.5 												:= FeedBwd;
	Status.6 												:= NOT Error;
	Status.7 												:= Error;
	
	(* Result *)
	_writeStatus											:= TRUE;
    												
(**************************************************************)
END_METHOD

{attribute 'monitoring' := 'call'}
PROPERTY public forwardStarted : BOOL
GET
forwardStarted := not Q_ContactorBwd and Q_Contactor;
END_GET
END_PROPERTY

{attribute 'monitoring' := 'call'}
PROPERTY public isOff : BOOL
GET
isOff := not Q_Contactor and not Q_ContactorBwd;
END_GET
END_PROPERTY

{attribute 'monitoring' := 'call'}
PROPERTY public isOn : BOOL
GET
isOn := Q_Contactor or Q_ContactorBwd;
END_GET
END_PROPERTY

{attribute 'monitoring' := 'call'}
PROPERTY noFeed : BOOL
GET
noFeed := NOT Feed and not FeedBwd;
END_GET
END_PROPERTY

{attribute 'monitoring' := 'call'}
PROPERTY public reverseStarted : BOOL
GET
reverseStarted := Q_ContactorBwd and not Q_Contactor;
END_GET
END_PROPERTY

METHOD PUBLIC startForward : bool //Return busy flag
VAR_INPUT
END_VAR
Start														:= TRUE;
StartBwd  := Q_ContactorBwd									:= FALSE;
Q_Contactor													:= ProtSwitchOK.Q AND Feed;
startForward												:= Q_Contactor;
Busy														:= startForward;
Error														:= NOT ProtSwitchOK.Q;
END_METHOD

METHOD PUBLIC startReverse : bool //Return busy flag
VAR_INPUT
END_VAR
StartBwd 													:= TRUE;
Start  := Q_Contactor										:= FALSE;
Q_ContactorBwd 												:= ProtSwitchOK.Q AND FeedBwd;
startReverse												:= Q_ContactorBwd;
Busy														:= startReverse;
Error														:= NOT ProtSwitchOK.Q;
END_METHOD

METHOD PUBLIC switchOff : BOOL //Return true if stopped / busy = false
VAR_INPUT
END_VAR
Start := startBwd											:= FALSE;
Q_Contactor := Q_ContactorBwd 								:= FALSE;
Busy														:= FALSE;
Error														:= NOT ProtSwitchOK.Q;
switchOff													:= TRUE;
END_METHOD

METHOD PUBLIC switchOn : BOOL  //True if motor is switched on
VAR_INPUT
END_VAR
switchOn := startForward();
END_METHOD

END_FUNCTION_BLOCK

// ---- POUs/IO/Motors/IOMotorStarDelta.TcPOU
{attribute 'no_check'}
FUNCTION_BLOCK IOMotorStarDelta EXTENDS IOMotor
VAR_INPUT
	PT_RestartDel											:	TIME := T#0S; //Delay to restart motor to avoid over heating
	PT_Delta												: 	TIME := T#5S; 
	ProtSwitchOK2											: 	FUSE;
END_VAR                 						
VAR_OUTPUT              						
	Q_StarContactor									AT %Q* 	: 	BOOL;
	Q_DeltaContactor								AT %Q* 	: 	BOOL;
	RestartDelActive										:	BOOL;
	ET_RestartDel											: 	TIME;	(* waiting-time of start interlock *)
END_VAR                 						
VAR                     						
	TON_StarDelta											:	TON;
	TP_RestartDel											:	TP;
END_VAR

(* Start Delta Motor IO	 				 	V1.1	*)
(****************************************************)

(* Protection Switch *****************************************)
	IF ResetTrig  THEN reset(); END_IF

	ProtSwitchOK();
	ProtSwitchOK2();
	
(* Start ****************************************************)
	IF Start THEN
		switchOn();
                       										
		Q_StarContactor 									:= 	Q_Contactor
																AND NOT TON_StarDelta.Q
																AND NOT Q_DeltaContactor;

		Q_DeltaContactor 									:= 	Q_Contactor
																AND TON_StarDelta.Q;

		TP_RestartDel();
	ELSE
		switchOff();
	END_IF

(* Timer *****************************************************)
	TON_StarDelta(IN := Q_Contactor, PT := PT_Delta);

	//Restart delay
	TP_RestartDel(IN := TP_RestartDel.Q,PT := PT_RestartDel); //Execute restart delay
	RestartDelActive										:= TP_RestartDel.Q;
	
	IF TP_RestartDel.ET > T#0MS 
	THEN
		ET_RestartDel		:= TP_RestartDel.PT - TP_RestartDel.ET;
	ELSE
		ET_RestartDel		:= t#0ms;
	END_IF
	
(* HMI status *********************************************)
	_writeStatus();
	
(********************************************************)

METHOD PROTECTED _writeStatus : BOOL
VAR_INPUT
END_VAR
(* HmiStatus **************************************************)
	Status.0												 := NOT Q_Contactor;
	Status.1												 := Q_Contactor;
	Status.2												 := Q_DeltaContactor;
	Status.3												 := RestartDelActive;
	Status.4												 := FALSE;
	Status.5												 := Feed;
	Status.6												 := NOT Error AND NOT RestartDelActive;
	Status.7												 := Error;

	(* Result *)
	_writeStatus											:= TRUE;
    												
(**************************************************************)
END_METHOD

{attribute 'monitoring' := 'call'}
PROPERTY public isOn : BOOL
GET
isOn := Q_Contactor;
END_GET
END_PROPERTY

{attribute 'monitoring' := 'call'}
PROPERTY ok : bool
GET
ok := Q_Contactor and Q_DeltaContactor ;
END_GET
END_PROPERTY

METHOD PUBLIC reset : booL
VAR_INPUT
END_VAR

reset									:= ProtSwitchOK.reset() AND ProtSwitchOK2.reset();
Error									:= FALSE;
END_METHOD

METHOD PUBLIC resetRestartTmr : booL
VAR_INPUT
END_VAR
MEMSET(ADR(TP_RestartDel),0,SIZEOF(TP_RestartDel));
resetRestartTmr										:= TRUE;
END_METHOD

METHOD public switchOff : BOOL
VAR_INPUT
END_VAR
Start														:= FALSE;
TP_RestartDel(IN := Q_Contactor , PT := PT_RestartDel);
Q_Contactor 												:= FALSE;
Q_StarContactor												:= FALSE;
Q_DeltaContactor											:= FALSE;
Busy														:= FALSE;
Error														:= NOT ProtSwitchOK.Q OR NOT ProtSwitchOK2.Q;
switchOff													:= TRUE;
END_METHOD

METHOD public switchOn : BOOL //True if motor is switched on
VAR_INPUT
END_VAR
Start														:= TRUE;
Q_Contactor		 											:= ProtSwitchOK.Q AND ProtSwitchOK2.Q AND Feed AND NOT TP_RestartDel.Q;
switchOn													:= Q_Contactor;
Busy														:= switchOn;
Error														:= NOT ProtSwitchOK.Q OR NOT ProtSwitchOK2.Q;
END_METHOD

END_FUNCTION_BLOCK

// ---- POUs/IpcDiag/MDP/InfoModuls/MDP_RaidSimple.TcPOU
{attribute 'no_check'}
FUNCTION_BLOCK MDP_RaidSimple  EXTENDS FbBase
VAR_OUTPUT CONSTANT
	MIN_DRIVE												:	INT := 1;
	MAX_DRIVE												:	INT := 4;
	                    									
//Cntr state            									
	CS_UNKNOWN												:	INT := 0;
	CS_GOOD													:	INT := 1;
	CS_FAILED												:	INT := 2; 
	CS_OFFLINE												:	INT := 3; 
	CS_POWER_OFF											:	INT := 4;
	                    									
//Cntr offline reason   									
	COR_NO_REASON											:	INT := 0;
	COR_INITIALIZING										:	INT := 1;
	COR_BUS_DEGRADED										:	INT := 2;
	COR_BUS_FAILURE											:	INT := 3;
	                    									
//Set state             									
	SS_OK													:	INT := 0;
	SS_DEGRADED												:	INT := 1;
	SS_REBUILDING											:	INT := 2;
	SS_FAILED												:	INT := 3;
	                    									
//Drive state		    									
	DS_OK													:	INT := 0;
	DS_REBUILDING											:	INT := 1;
	DS_FAILED 												:	INT := 2;
	DS_DEGRADED 											:	INT := 3;
END_VAR                 									
VAR_INPUT               									
	AmsNetId												: 	T_AmsNetId := '';	//AmsNetId as text
	Timeout													:	TIME := DEFAULT_ADS_TIMEOUT;	//Ads timeout
END_VAR                 									
VAR_OUTPUT              									
(* Raid Data *)         									
	CntrState												:	INT := CS_UNKNOWN;		//current controller state
	CntrOfflReason 											: 	INT := COR_NO_REASON;	//reason for controller offline
                        									
	SetType													:	USINT;					//type of RAID system
	SetState												:	INT := SS_OK;			
	SetInfo													:	USINT; (* 	If SetStatus = OK, THEN Info will be 0.
																					If SetStatus = DEGRADED, then Info will contain the failed drive index number.1
																					If SetStatus = REBUILDING, then Info will contain the percentage complete. The value will be in the range of 0 to 100 (0h to 64h).
																					If SetStatus == FAILED, then Info will be 0 or vendor specific. Since the failure modes could include drive or controller failures, Info may provide a vendor specific error code to indicate which component led to the failed status. *)
	CountDrives												:	UINT;
	DriveSTATE												:	ARRAY[MIN_DRIVE..MAX_DRIVE] OF INT; //current state of drive
	CountRAIDSets											:	UINT; 		//Count RAID sets
	ErrorGrp												:	E_MDP_ErrGroup := eMDP_Err_NoError;
END_VAR                 									
VAR                     									
	idx														:	INT := 1;
	MDP_ScanModules											:	FB_MDP_ScanModules := ( nModuleType 	:= eMDP_ModT_RAID , iModIdx		:= 0);
	MDP_Read												: 	FB_MDP_Read;
	SplitErrorId											:	FB_MDP_SplitErrorID ;
	DstBuf													:	ARRAY[0..4] OF BYTE;
END_VAR

(* Read RAID Information 						V1.0	*)
(* only for RAID set 1									*)
(* not more then MAX_DRIVES per RAID set				*)
(********************************************************)

(* Start Read *******************************************)
	IF Execute
		AND state = 0
	THEN
		CntrState											:= CS_UNKNOWN;
		CntrOfflReason 										:= COR_NO_REASON;
		SetType												:= 0;
		SetState											:= SS_OK;
		SetInfo												:= 0;
		CountDrives											:= 0;
		MEMSET(ADR(DriveSTATE),0,SIZEOF(DriveSTATE));   	
		CountRAIDSets										:= 0;
                                                        	
		Busy												:= TRUE;
		Done												:= FALSE;
		Error												:= FALSE;
		ErrorId												:= 0;
		ErrorGrp											:= eMDP_Err_NoError;
		MDP_Read(bExecute := FALSE);
		MDP_ScanModules(
			bExecute		:= FALSE,
			nModuleType		:= eMDP_ModT_RAID,
			iModIdx			:= 0,
			tTimeout		:= timeout,
			sAmsNetId		:= AmsNetId,
			bBusy			=> ,
			bError			=> ,
			nErrID			=> ,
			nDynModuleId	=> ,
			iModuleTypeCount=> ,
			iModuleCount	=> );
			
		MDP_ScanModules(bExecute:= TRUE);
		state												:= 1;
	ELSIF NOT Execute
		AND State = 99
	THEN
		state												:= 0;
		Busy												:= FALSE;
		Done												:= FALSE;
		Error												:= FALSE;
		ErrorId												:= 0;
		ErrorGrp											:= eMDP_Err_NoError;
	END_IF


	CASE state OF
	0:
		;
	1:
		MDP_ScanModules();
		IF NOT MDP_ScanModules.bBusy
		THEN
			IF MDP_ScanModules.bError
			THEN
				Busy										:= FALSE;
				Error										:= TRUE;
				SplitErrorId(
					nErrID		:= MDP_ScanModules.nErrID,
					eErrGroup	=> ErrorGrp ,
					nErrCode	=> ErrorId);
				state										:= 99;
				MDP_ScanModules(bExecute := FALSE);
			ELSE
				MDP_Read(bExecute := FALSE);
				MDP_Read.stMDP_DynAddr.nArea				:= 16#8;
				MDP_Read.stMDP_DynAddr.nModuleId			:= MDP_ScanModules.nDynModuleId;
				MDP_Read.stMDP_DynAddr.nTableId				:= 16#1;
				MDP_Read.stMDP_DynAddr.nSubIdx				:= 0;
				state										:= 2;
			END_IF

		END_IF

	2:
		MDP_Read( pDstBuf	:= ADR(DstBuf), cbDstBufLen := SIZEOF(DstBuf));
		IF NOT MDP_Read.bBusy
		THEN
			IF MDP_Read.bError AND MDP_Read.bExecute
			THEN
				IF MDP_Read.stMDP_DynAddr.nTableId = 16#2
					AND MDP_Read.stMDP_DynAddr.nSubIdx = 1
				THEN (* No RaidSystem found *)
					Busy									:= FALSE;
					Done									:= TRUE;
					state									:= 99;
				ELSE
					Busy									:= FALSE;
					Error									:= TRUE;
					SplitErrorId(
						nErrID		:= MDP_Read.nErrID,
						eErrGroup	=> ErrorGrp ,
						nErrCode	=> ErrorId);
				END_IF
				state										:= 99;
				MDP_Read(bExecute := FALSE);
			ELSE
				MDP_Read(bExecute := FALSE);
				CASE MDP_Read.stMDP_DynAddr.nTableId OF
				16#1: (* Controller Info *)
					CASE MDP_Read.stMDP_DynAddr.nSubIdx	OF
					0:
						MDP_Read.stMDP_DynAddr.nSubIdx		:= 1;

					1:
						MEMCPY(ADR(CntrState), ADR(DstBuf), SIZEOF(CntrState));
						MDP_Read.stMDP_DynAddr.nSubIdx		:= 2;

					2:
						MEMCPY(ADR(CntrOfflReason), ADR(DstBuf), SIZEOF(CntrOfflReason));
						MDP_Read.stMDP_DynAddr.nSubIdx		:= 0;
						MDP_Read.stMDP_DynAddr.nTableId		:= 16#2;
					END_CASE

				16#2: (* Raid Sets Type *)
					CASE MDP_Read.stMDP_DynAddr.nSubIdx	OF
					0:
						MEMCPY(ADR(CountRAIDSets), ADR(DstBuf), SIZEOF(CountRAIDSets));
						MDP_Read.stMDP_DynAddr.nSubIdx		:= 1;

					1:
						MEMCPY(ADR(SetType), ADR(DstBuf), SIZEOF(SetType));
						MDP_Read.stMDP_DynAddr.nSubIdx		:= 1;
						MDP_Read.stMDP_DynAddr.nTableId		:= 16#3;
					END_CASE

				16#3: (* RAID sets state and info *)
					CASE MDP_Read.stMDP_DynAddr.nSubIdx	OF
					1:
						MEMCPY(ADR(SetState), ADR(DstBuf[0]), 1);
						MEMCPY(ADR(SetInfo), ADR(DstBuf[1]), 1);
						MDP_Read.stMDP_DynAddr.nSubIdx		:= 0;
						MDP_Read.stMDP_DynAddr.nTableId		:= 16#A;
					END_CASE


				16#A: (* Drives state  *)
					CASE MDP_Read.stMDP_DynAddr.nSubIdx	OF
					0:
						MEMCPY(ADR(CountDrives), ADR(DstBuf), SIZEOF(CountDrives));
						MDP_Read.stMDP_DynAddr.nSubIdx		:= 1;

					1..255:
						MEMCPY(ADR(DriveSTATE), ADR(DstBuf), 1);
						MDP_Read.stMDP_DynAddr.nSubIdx	:= MDP_Read.stMDP_DynAddr.nSubIdx + 1;
						IF MDP_Read.stMDP_DynAddr.nSubIdx > CountDrives
							OR MDP_Read.stMDP_DynAddr.nSubIdx > MAX_DRIVE
						THEN
							Busy							:= FALSE;
							Done							:= TRUE;
							state							:= 99;
						END_IF

					END_CASE

				ELSE
					Busy									:= FALSE;
					Done									:= TRUE;
					state									:= 99;
				END_CASE

				MDP_Read(
					stMDP_DynAddr	:= ,(* address to request subindex Count of AdressList *)
					pDstBuf			:= ADR(DstBuf),
					cbDstBufLen		:= SIZEOF(DstBuf),
					bExecute		:= NOT MDP_Read.bBusy AND state = 2,
					tTimeout		:= Timeout,
					sAmsNetId		:= AmsNetId,
					bBusy			=> ,
					bError			=> ,
					nErrId			=> );
			END_IF
		END_IF

	99: ;

	ELSE
		;
	END_CASE

	(* reset state for next start *)
	IF NOT Execute
		AND state = 99
	THEN
		state												:= 0;
	END_IF

(****************************************************************************************************)

END_FUNCTION_BLOCK

// ---- POUs/Logging/Logbook.TcPOU
{attribute 'no_check'}
//PLC Logbook for debugging, records a number of "MAX_DATA" messages with timestamp.
//The Logbook Puplisher can be used to forward messages from the logbook to several subscriber (Write into Logfile, display via EventLogger, send to Syslog Server)
//
//Parameter Timestamp needs to be updated externaly every cycle if needed
//
//Function "LogWithEventClass" is used inside
FUNCTION_BLOCK Logbook IMPLEMENTS I_Logbook                 									
VAR_OUTPUT CONSTANT     									
//Parameter
	MIN_DATA												:	INT := 1;
	MAX_DATA												:	INT := PARAM.LOGBOOK_MAX_DATA; //see library parameter to customize parameter	
                        									
//option settings to modify the message string and behavior
{attribute 'displaymode':='binary'}
	OPTION_WRITE_TO_ADSLOG									: 	BYTE :=2#0000_0100; //Write entry directly to TwinCAT logger (shown in XAE output)
{attribute 'displaymode':='binary'}
	OPTION_ADD_TIME_TO_MSG_STRING							: 	BYTE :=2#0000_1000;	//Add time stamp to message string 
{attribute 'displaymode':='binary'}
	OPTION_ADD_DATE_TO_MSG_STRING							: 	BYTE :=2#0001_0000; //Add date to message string
END_VAR                 									
VAR_INPUT               									                       		
{attribute 'displaymode':='binary'}
	Options													:	BYTE := 2#0000_0000;			(* option constants are alreay predefined, so they can accordingly be passed symbolically to the block
																								Bit 0 = 
																								Bit 1 = 
																								Bit 2 = Send to TC Ads-Logger
																								Bit 3 = Add time to message string
																								Bit 4 = Add date to message string
																								Bit 5 = 
																								Bit 6 = 
														 										Bit 7 =  								
																								*)
                        									
// InputData         	
	Timestamp												:	TIMESTRUCT; //Time stamp need to be updated cylic if it will be used
	Msg														:	STRING(PARAM.LOGBOOK_MAX_MSG_STRING_LENGHT) := ''; //Message string which will written into the DataMsg array by executing the Fb																							
END_VAR             										
VAR_OUTPUT
	Data													:	ARRAY[MIN_DATA..MAX_DATA] OF LogbookData; // Recorded messages data
	CntAddedMessages										:	INT;
END_VAR
VAR
	TaskInterlock											:	BOOL;
END_VAR

(* LogBook 									 *)
(*********************************************)

(* call method *********************************************)
	_Write(Msg);
(***********************************************************)

METHOD PROTECTED _write : BOOL
VAR_IN_OUT
	Msg														:	STRING(PARAM.LOGBOOK_MAX_MSG_STRING_LENGHT);
END_VAR
(* Write entry with every call ******************************)
IF LEN(MSG) = 0
THEN
	_Write													:= FALSE;
	RETURN;
ELSIF TestAndSet(TaskInterlock)
THEN	
	MEMMOVE(ADR(Data[MIN(MIN_DATA + 1,MAX_DATA)]), 	ADR(Data), 	SIZEOF(Data) - SIZEOF(Data[MIN_DATA]));
	
	(* Datensatz oben eintragen *)
	IF NOT Options.3 AND NOT Options.4
	THEN
		Data[MIN_DATA].Msg									:= Msg;
	ELSIF Options.3 AND Options.4              
	THEN                                                    
		Data[MIN_DATA].Msg									:= SYSTEMTIME_TO_STRING(Timestamp);
		Data[MIN_DATA].Msg									:= CONCAT(Data[MIN_DATA].Msg, ' | ');
		Data[MIN_DATA].Msg									:= CONCAT(Data[MIN_DATA].Msg, Msg);
	ELSIF Options.4                                   
	THEN                                                    
		Data[MIN_DATA].Msg									:= SYSTEMTIME_TO_STRING(Timestamp);
		Data[MIN_DATA].Msg									:=	MID(Data[MIN_DATA].Msg, 12 , 12);
		Data[MIN_DATA].Msg									:= CONCAT(Data[MIN_DATA].Msg, ' | ');
		Data[MIN_DATA].Msg									:= CONCAT(Data[MIN_DATA].Msg, Msg);
                                                            
	ELSE (* Only Date to Msg String *)                      
		Data[MIN_DATA].Msg									:= SYSTEMTIME_TO_STRING(Timestamp);
		Data[MIN_DATA].Msg									:= MID(Data[MIN_DATA].Msg, 8 , 3);
		Data[MIN_DATA].Msg									:= CONCAT(Data[MIN_DATA].Msg, ' | ');
		Data[MIN_DATA].Msg									:= CONCAT(Data[MIN_DATA].Msg, Msg);
	END_IF                                                  

	//Coyp current options from logbook into message	                                                        
	Data[MIN_DATA].Options									:= TO_WORD(Options);
		
	//Store time stamp
	Data[MIN_DATA].Timestamp								:= Timestamp;
	
	CntAddedMessages										:= MIN(MAX_DATA, CntAddedMessages + 1); 
	_Write													:= TRUE;
	TaskInterlock											:= FALSE;
END_IF

(************************************************************)
END_METHOD

METHOD PUBLIC delete : BOOL //Return value = TRUE if execution finished
VAR_INPUT
END_VAR

CntAddedMessages											:= 0;
MEMSET(ADR(Data),0,SIZEOF(Data));
delete														:= TRUE;
END_METHOD

METHOD PUBLIC getOldestMsg : BOOL //Return value TRUE = if finished successful -> new message read
VAR_IN_OUT
	data													: LogbookData;								
END_VAR
IF CntAddedMessages >= MIN_DATA AND CntAddedMessages <= MAX_DATA
	AND NOT TaskInterlock
THEN
	data													:= THIS^.Data[CntAddedMessages];
	THIS^.Data[CntAddedMessages].Options.15					:= FALSE; //New message
	CntAddedMessages										:= CntAddedMessages - 1;
	getOldestMsg											:= TRUE;
ELSE
	getOldestMsg											:= FALSE;
END_IF
END_METHOD

PROPERTY PUBLIC optAddDateToMsgText : BOOL
GET
optAddDateToMsgText := Options.4;
END_GET
SET
Options.4 := optAddDateToMsgText;
END_SET
END_PROPERTY

PROPERTY PUBLIC optAddTimeToMsgText : BOOL
GET
optAddTimeToMsgText := Options.3;
END_GET
SET
Options.3 := optAddTimeToMsgText;
END_SET
END_PROPERTY

PROPERTY Public optWiteEntryToTcAdsLogger : BOOL
GET
optWiteEntryToTcAdsLogger := Options.2;
END_GET
SET
Options.2 := optWiteEntryToTcAdsLogger;
END_SET
END_PROPERTY

{attribute 'monitoring' := 'call'}
PROPERTY PUBLIC rCntAddedMessages : Reference to INT //Reference to variable showing no of added messages (Counter will be decreased by getOldestMsg)
GET
rCntAddedMessages REF= CntAddedMessages;
END_GET
END_PROPERTY

METHOD PUBLIC readMsg : REFERENCE TO LogbookData //Return value is a REFERENCE to the by Index selected entry.  
VAR_INPUT
	Index											:	INT;						
END_VAR

readMsg													REF= THIS^.Data[LIMIT(MIN_DATA,Index,MAX_DATA)];
END_METHOD

METHOD PUBLIC write : BOOL //Return value = TRUE if execution finished
VAR_INPUT
	Msg														:	STRING(PARAM.LOGBOOK_MAX_MSG_STRING_LENGHT);
END_VAR

write														:= _Write(Msg);
IF options.2 
THEN
	write 													:= write AND 0 = adsLogHint(Msg, '');
END_IF
END_METHOD

END_FUNCTION_BLOCK

// ---- POUs/Motion/TF50xx-NC/03_Utilities/CoordinateTransformation2D.TcPOU
FUNCTION_BLOCK CoordinateTransformation2D //CoordinateTransformation
// transformation of an X/Y product coordinate to the machine coordinate system
// MCS = machine coordinate system
// PCS = product coordinate system
VAR_INPUT
//Parameter
	x0 														: LREAL;		// origin MCS X coordinate of the product coordinate system
	y0 														: LREAL;		// origin MCS Y coordinate of the product coordinate system
	x1 														: LREAL;		// opposite corner point MCS X coordinate of the product 
	y1 														: LREAL;		// opposite corner point MCS Y coordinate of the product
	a 														: LREAL;		// length of the product (difference x1pcs-x0pcs)
	b 														: LREAL;		// width of the product (difference y1pcs-y0pcs)
END_VAR                                                 	
VAR_OUTPUT                                              	
	Xmcs 													: LREAL;	// X coordinate in machine coordinate system
	Ymcs 													: LREAL;	// Y coordinate in machine coordinate system
															
	Xpcs 													: LREAL;	// X coordinate in Product coordinate system
	Ypcs 													: LREAL;	// Y coordinate in Product coordinate system
                                                        	
	Alfa													: LREAL;	

	Error 													: BOOL;	
//		ErrorID 											: UDINT;
END_VAR
VAR
	c														: LREAL;
	diagonal												: LREAL;

	ratio													: LREAL;
	
	alfa1													: LREAL;
	alfa2													: LREAL;
END_VAR

;

{attribute 'monitoring' := 'call'}
PROPERTY PUBLIC diagonalMSC : LREAL
GET
VAR
	t		:	LREAL;
END_VAR
t 			:=  EXPT(X1-X0,2.0) + EXPT(y1-y0,2.0);
DiagonalMSC := SQRT(t);
END_GET
END_PROPERTY

{attribute 'monitoring' := 'call'}
PROPERTY PUBLIC diagonalPCS : LREAL
GET
DiagonalPCS := SQRT((a*a)+(b*b));
END_GET
END_PROPERTY

{attribute 'monitoring' := 'call'}
PROPERTY PUBLIC isParamValid : BOOL
GET
IsParamValid 													:= not ParamHasError;
END_GET
SET // PUBLIC
IF NOT IsParamValid
THEN
	a 														:= 0.0;
	b 														:= 0.0;
	x1 														:= Y1 := 0.0;
	y0 														:= X0 := 0.0;
END_IF
END_SET
END_PROPERTY

METHOD MSCtoPCS : BOOL //Return value = TRUE if execution finished successful / FALSE if finished with error
VAR_INPUT
	Xmcs 													: LREAL;	// X coordinate in machine coordinate system
	Ymcs 													: LREAL;	// Y coordinate in machine coordinate system
END_VAR
IF ParamHasError THEN
	Error 													:= TRUE; 
	MSCtoPCS 												:= FALSE;
ELSE	
	THIS^.Xmcs												:= Xmcs;	
	THIS^.Ymcs												:= Ymcs;	

	c 														:= SQRT(a*a + b*b);
	alfa 													:= ACOS((x1-x0) / c) - ACOS( a / c);
	
	Xpcs 													:= 	 (Xmcs - x0) * COS(alfa) + (Ymcs - y0) * SIN(alfa);
	Ypcs 													:= - (Xmcs - x0) * SIN(alfa) + (Ymcs - y0) * COS(alfa);
	
	Error 													:= FALSE; 
	MSCtoPCS 												:= TRUE;
END_IF
END_METHOD

{attribute 'monitoring' := 'call'}
PROPERTY PRIVATE paramHasError : BOOL
GET
ParamHasError := 	a<=0.0 
			OR 	b<=0.0 
			OR 	x1=x0 
			OR 	y1=y0;
END_GET
END_PROPERTY

METHOD PUBLIC PCStoMSC : booL //Return value = TRUE if execution finished successful / FALSE if finished with error
VAR_INPUT
	Xpcs : LREAL;	// X coordinate in product coordinate system
	Ypcs : LREAL;	// Y coordinate in product coordinate system	
END_VAR
IF ParamHasError 
THEN
	Error 													:= TRUE; 
	PCStoMSC												:= FALSE;
ELSE                										
	THIS^.Xpcs												:= Xpcs;	
	THIS^.Ypcs												:= Ypcs;
	
	c 														:= SQRT(a*a + b*b);
	diagonal												:= SQRT((x1-x0)*(x1-x0)+(y1-y0)*(y1-y0));
	
	ratio													:= diagonal/c;
	
	alfa1 													:= ACOS((x1-x0) / diagonal);
	alfa2													:= ACOS(a/c);
	
	alfa													:= alfa1-alfa2;
	
	Xmcs 													:= x0 + ratio * (Xpcs * COS(alfa) - Ypcs * SIN(alfa));
	Ymcs 													:= y0 + ratio * (Xpcs * SIN(alfa) + Ypcs * COS(alfa));
                    	
	Error 													:= FALSE; 
	PCStoMSC												:= TRUE;
END_IF
END_METHOD

END_FUNCTION_BLOCK

// ---- POUs/Motion/TF50xx-NC/AxNcPTPwJobs.TcPOU
FUNCTION_BLOCK AxNcPTPwJobs EXTENDS AxNcPTP (* See Tc2_MC2 *)
VAR_OUTPUT CONSTANT
	MIN_JOB													:	INT := 0;
	MAX_JOB													:	INT := 5;
	
{attribute 'displaymode':='binary'}
	OPTION_EN_CYCLIC_TARGET_CHECK							: 	BYTE := 2#0000_0001; //.0 = Cyclic target check	
END_VAR
VAR_INPUT
	Job														:	ARRAY[MIN_JOB..MAX_JOB] OF AX_JOB;	                              
END_VAR                           
var_output                  	
	JobId													:	INT := MIN_JOB;
END_VAR
VAR
	i 														: 	INT;
END_VAR

	(* Axis 																*)
	(************************************************************************)

	
(********************************************************************************)
(* Call AxNcBase																*)
(********************************************************************************)
	Super^();
			
(* Check start arr pos **********************************************************)
	IF Options.0 AND Para.InitDone THEN	CheckTargetPos(); END_IF
	
(********************************************************************************)

METHOD PUBLIC checkTargetPos : INT //ID of last job which is in target / 0 if no job is in target
VAR_INPUT
END_VAR
CheckTargetPos				:= 0;
FOR i := MIN_JOB TO MAX_JOB DO
	IF Job[i].Fnc = 6 THEN
		Job[i].InTarget := Status.NotMoving
									AND(
									NcToPlc.ModuloActPos >= Job[i].Target - para.TargetPosWindow
									AND NcToPlc.ModuloActPos <= Job[i].Target + para.TargetPosWindow
									OR
									(MODABS(Job[i].Target,para.ModuloFactor) <= 0 + para.TargetPosWindow
									OR MODABS(Job[i].Target,para.ModuloFactor) >= para.ModuloFactor - para.TargetPosWindow)
									AND(
									NcToPlc.ModuloActPos >= para.ModuloFactor - para.TargetPosWindow
									OR NcToPlc.ModuloActPos <= 0 + para.TargetPosWindow));

		Job[i].InPosWindow	:= NcToPlc.ModuloActPos >= Job[i].Target - para.PosRangeWindow
									AND NcToPlc.ModuloActPos <= Job[i].Target + para.PosRangeWindow
									OR
									(MODABS(Job[i].Target,para.ModuloFactor) <= 0 + para.PosRangeWindow
									OR MODABS(Job[i].Target,para.ModuloFactor) >= para.ModuloFactor - para.PosRangeWindow)
									AND(
									NcToPlc.ModuloActPos >= para.ModuloFactor - para.PosRangeWindow
									OR NcToPlc.ModuloActPos <= 0 + para.PosRangeWindow);
	ELSE
		Job[i].InTarget := Status.NotMoving
									AND NcToPlc.ActPos >= Job[i].Target - para.TargetPosWindow
									AND NcToPlc.ActPos <= Job[i].Target + para.TargetPosWindow ;

		Job[i].InPosWindow	:= NcToPlc.ActPos >= Job[i].Target - para.PosRangeWindow
									AND NcToPlc.ActPos <= Job[i].Target + para.PosRangeWindow;
	END_IF
	
	IF Job[i].InTarget 
	THEN
		CheckTargetPos		:= i;
	END_IF
END_FOR
END_METHOD

PROPERTY PUBLIC optEnableCyclicCheckTargetPos : BOOL
GET
optEnableCyclicCheckTargetPos := Options.0;
END_GET
SET
Options.0 := optEnableCyclicCheckTargetPos;
END_SET
END_PROPERTY

METHOD PUBLIC startMotion : BOOL
VAR_INPUT
	Execute			:	BOOL;
	JobID			:	int ;
END_VAR
THIS^.JobID		:= Jobid;

IF JobID >= MIN_JOB AND JobId <= MAX_JOB
THEN
	CheckTargetPos();
//	startName				:= Job[Jobid].name;
	Motion.Fnc 				:= Job[Jobid].Fnc;
	Motion.BufferMode 		:= Job[Jobid].BufferMode;
	Motion.Direction 		:= Job[Jobid].Direction;
	Motion.Target 			:= Job[Jobid].Target;
	Motion.Velo 			:= Job[Jobid].Velo;
	Admin.Override 			:= Job[Jobid].Override;
	Motion.Acc		 		:= Job[Jobid].Acc;
	Motion.Dec				:= Job[Jobid].Dec;
	Motion.Jerk	 			:= Job[Jobid].Jerk;
	MOtion.Execute			:= Execute;
	StartMotion				:= TRUE;
ELSE
	StartMotion				:= FALSE;
END_IF
END_METHOD

END_FUNCTION_BLOCK

// ---- POUs/Motion/TF511x-KIN/03_DUTs/Trafo/KIN_STATICTRAFO_PARAM.TcPOU
{attribute 'hide'}
FUNCTION_BLOCK KIN_STATICTRAFO_PARAM
VAR_INPUT
	oid														:	UDINT := 0;
	TranslationX											:	LREAL := 0.0;
	TranslationY											:	LREAL := 0.0;
	TranslationZ											:	LREAL := 0.0;
                            								
	Rotation												: LREAL := 0.0;
	RotationAxis											: INT := 2;

END_VAR
VAR_OUTPUT

END_VAR
VAR
END_VAR

;

METHOD delete : BOOL
VAR_INPUT
END_VAR
	oid														:= 0;
	TranslationX											:= 0.0;
	TranslationY											:= 0.0;
	TranslationZ											:= 0.0;
                            								
	Rotation												:= 0.0;
	RotationAxis											:= 2;
delete	:= TRUE;
END_METHOD

END_FUNCTION_BLOCK

// ---- POUs/Motion/TF511x-KIN/03_DUTs/Trafo/UCS.TcPOU
{attribute 'hide'}
FUNCTION_BLOCK UCS
VAR_INPUT
	oid														:	UDINT := 0;		//Object identifier
	vTranslation 											:	VECTOR;
 	vRotation 												:	VECTOR;
	Valid													:	BOOL := FALSE;
END_VAR
VAR_OUTPUT
END_VAR
VAR
END_VAR

METHOD delete : BOOL
VAR_INPUT
END_VAR
MEMSET(ADR(vTranslation),0,SIZEOF(vTranslation));
MEMSET(ADR(VRotation),0,SIZEOF(VRotation));
oid 													:= 0;
delete	:= TRUE;
END_METHOD

END_FUNCTION_BLOCK

// ---- POUs/Motion/VALUE_3D.TcPOU
{attribute 'no_check'}
FUNCTION_BLOCK VALUE_3D
VAR_INPUT                                                            
	Valid													:	BOOL ;
	X														:	LREAL;
	Y														:	LREAL;
	Z														:	LREAL;
END_VAR
VAR_OUTPUT
END_VAR
VAR
END_VAR

;

METHOD PUBLIC copy : BOOL //Return value = TRUE if execution finished
VAR_IN_OUT
	Source													:	VALUE_3D;
END_VAR
	Valid													:= Source.Valid;
	X														:= Source.X;
	Y														:= Source.Y;
	Z														:= Source.Z;
	copy													:= TRUE;
END_METHOD

METHOD PUBLIC delete : BOOL //Return value = TRUE if execution finished - Valid bit will not change
VAR_INPUT
END_VAR
	X					 									:= 0.0;	
	Y					 									:= 0.0;	
	Z					 									:= 0.0;	
	delete													:= TRUE;
END_METHOD

METHOD PUBLIC InPos : BOOL //Return value = TRUE axes is within window of checkPos values
VAR_IN_OUT
	CheckPos												:	VALUE_3D;
	Window													:	VALUE_3D;
END_VAR
InPos														:= CAM(CheckPos.X, X ,Window.X)
																AND CAM(CheckPos.Y, Y ,Window.Y)
																AND CAM(CheckPos.Z, Z ,Window.Z);
END_METHOD

METHOD PUBLIC InPosByAxisNo : BOOL //Return value = TRUE selected axis is within window of checkPos values
VAR_INPUT
	No					:	INT;
END_VAR
VAR_IN_OUT
	CheckPos			:	VALUE_3D;
	Window				:	VALUE_3D;
END_VAR
InPosByAxisNo													:= (CAM(CheckPos.X, X ,Window.X) OR No <> 1)
																AND (CAM(CheckPos.Y, Y ,Window.Y) OR No <> 2)
																AND (CAM(CheckPos.Z, Z ,Window.Z) OR No <> 3);
END_METHOD

METHOD PUBLIC InPosXY : BOOL //Return value = TRUE if axes are within window of checkPos values
VAR_IN_OUT
	CheckPos			:	VALUE_3D;
	Window				:	VALUE_3D;
END_VAR
InPosXY 													:= CAM(CheckPos.X, X ,Window.X)
																AND CAM(CheckPos.Y, Y ,Window.Y);
END_METHOD

METHOD PUBLIC InPosXZ : BOOL //Return value = TRUE if axes are within window of checkPos values
VAR_IN_OUT
	CheckPos			:	VALUE_3D;
	Window				:	VALUE_3D;
	
END_VAR
InPosXZ														:= CAM(CheckPos.X, X ,Window.X)
																AND CAM(CheckPos.Z, Z ,Window.Z);
END_METHOD

METHOD PUBLIC InPosYZ : BOOL //Return value = TRUE if axes are within window of checkPos values
VAR_IN_OUT
	CheckPos			:	VALUE_3D;
	Window				:	VALUE_3D;
	
END_VAR
InPosYZ													:= CAM(CheckPos.Y, Y ,Window.Y)
																AND CAM(CheckPos.Z, Z ,Window.Z);
END_METHOD

METHOD PUBLIC reset : BOOL //Delete data and reset valid , TRUE if execution finished
VAR_INPUT
END_VAR
Delete();
Valid														:= FALSE;
reset														:= TRUE;
END_METHOD

END_FUNCTION_BLOCK

// ---- POUs/Safety/Diag/SafetyLogicAndIOTerminalDiag.TcPOU
{attribute 'no_check'}
FUNCTION_BLOCK SafetyLogicAndIOTerminalDiag EXTENDS SafetyLogicTerminalDiag
VAR_OUTPUT CONSTANT
	MIN_IN_MODULE											:	INT := 1;
	MAX_IN_MODULE											:	INT := Param.SAFETY_LOGIC_IO_TERM_DIAG_MAX_MODULE; 
	MIN_OUT_MODULE											:	INT := 1;
	MAX_OUT_MODULE											:	INT := Param.SAFETY_LOGIC_IO_TERM_DIAG_MAX_MODULE; 	
END_VAR                 									
VAR_INPUT               									
	FSOUT_Module_Output								AT %Q*	:	ARRAY[MIN_OUT_MODULE..MAX_OUT_MODULE] OF BOOL;	
END_VAR
VAR_OUTPUT
	FSIN_Module_Fault								AT %I*	:	ARRAY[MIN_IN_MODULE..MAX_IN_MODULE] OF BOOL;
	FSOUT_Module_Fault								AT %I*	:	ARRAY[MIN_OUT_MODULE..MAX_OUT_MODULE] OF BOOL;

END_VAR
VAR 
END_VAR
VAR 
(* Events/Blocks/Var internal *)
	EventFSINModuleFault									:	EventHandling := (SourceId := DEFAULT_SOURCE_ID, MsgId:= 7);	
	EventFSOUTModuleFault									:	EventHandling := (SourceId := DEFAULT_SOURCE_ID, MsgId:= 8);
	
{attribute 'displaymode':='binary'}
	FSIN_Faults												:	DWORD; 
{attribute 'displaymode':='binary'}
	FSOUT_Faults											:	DWORD; 

END_VAR

(* Extension to ELx9xx Safety Logic with local IO's Terminal Diag	*)
(********************************************************************)

(* call super *************************************************************)
	SUPER^();
	
(* Event 7-8 *******************************************************************)
	FOR i := MIN_IN_MODULE TO MAX_IN_MODULE
	DO
		FSIN_Faults											:= CSETBIT32(FSIN_Faults,TO_SINT(i-1),FSIN_Module_Fault[i]);
	END_FOR
		
	EventFSINModuleFault(
		Flag		:= FSIN_Faults <> 0 AND_THEN IO.InfoDataState = Tc2_EtherCAT.EC_DEVICE_STATE_OP AND Enable,
		ConfirmTrig	:= Quit OR NOT Enable,
		MsgId		:= ,
		SourceId	:= ,
		eClass		:=,
		format		:= ,
		Text1		:= DWORD_TO_BINSTR_EXT(FSIN_Faults,MAX_IN_MODULE,3),
		Text2		:= ,
		pText3		:= ADR(IO.DevName),
		State		=> ,
		Status		=> );

	FOR i := MIN_OUT_MODULE TO MAX_OUT_MODULE
	DO
		FSOUT_Faults											:= CSETBIT32(FSOUT_Faults,TO_SINT(i-1),FSOUT_Module_Fault[i]);
	END_FOR
			 	
	EventFSOUTModuleFault(
		Flag		:= FSOUT_Faults <> 0 AND_THEN IO.InfoDataState = Tc2_EtherCAT.EC_DEVICE_STATE_OP AND Enable,
		ConfirmTrig	:= Quit OR NOT Enable,
		MsgId		:= ,
		SourceId	:= ,
		eClass		:=,
		format		:= ,
		Text1		:= DWORD_TO_BINSTR_EXT(FSIN_Faults,MAX_OUT_MODULE,3),
		Text2		:= ,
		pText3		:= ADR(IO.DevName),
		State		=> ,
		Status		=> );	
				
	Status													:= Status OR EventFSINModuleFault.Status OR EventFSOUTModuleFault.Status;
(*****************************************************************)

{attribute 'monitoring' := 'call'}
PROPERTY PUBLIC inputModuleFault : bool
GET
VAR
	i	: int;
END_VAR
inputModuleFault									:= FALSE;
FOR i := MIN_IN_MODULE TO MAX_IN_MODULE
DO
	IF FSIN_Module_Fault[i]
	THEN
		inputModuleFault							:= TRUE;
		EXIT;
	END_IF
	
END_FOR
END_GET
END_PROPERTY

{attribute 'monitoring' := 'call'}
PROPERTY PUBLIC moduleInFault : bool
GET
moduleInFault			:= inputModuleFault or outputModuleFault;
END_GET
END_PROPERTY

{attribute 'monitoring' := 'call'}
PROPERTY PUBLIC outputModuleFault : bool
GET
VAR
	i : int;
END_VAR
outputModuleFault									:= FALSE;
FOR i := MIN_OUT_MODULE TO MAX_OUT_MODULE
DO
	IF FSOUT_Module_Fault[i]
	THEN
		outputModuleFault							:= TRUE;
		EXIT;
	END_IF
	
END_FOR
END_GET
END_PROPERTY

END_FUNCTION_BLOCK

// ---- POUs/_Miscellaneous/Conversions/DWORD_TO_REAL_EX.TcPOU
// Converts a 32bit float variable with swapped words into a TwinCAT conform REAL value after checking whether the result will be a valid number
// Use PDWORD_TO_DWORD in case the source variable is e..g a byte array -> RealVar := DWORD_TO_REAL_EX(In := PDWORD_TO_DWORD(ADR(ModBusCom.Data[1]));
FUNCTION DWORD_TO_REAL_EX : REAL
VAR_INPUT
	In						:	DWORD;
END_VAR
VAR
	Dummy					: U_32BIT_DATATYPE;
END_VAR


	Dummy._DWORD			:= In;

	F_SwapRealEx(Dummy._REAL);

	IF	IsFinite(F_REAL(Dummy._REAL)) THEN
		DWORD_TO_REAL_EX := Dummy._REAL;
	ELSE
		DWORD_TO_REAL_EX := 0.0;
	END_IF

END_FUNCTION

// ---- POUs/_Miscellaneous/Conversions/LWORD_TO_LREAL_EX.TcPOU
// Converts a 64bit double variable with swapped words into a TwinCAT conform LREAL value after checking whether the result will be a valid number
// Use PLWORD_TO_LWORD in case the source variable is e..g a byte array -> LRealVar := LWORD_TO_LREAL_EX(In := PLWORD_TO_LWORD(ADR(ModBusCom.Data[1]));
FUNCTION LWORD_TO_LREAL_EX : LREAL
VAR_INPUT
	In						: LWORD;
END_VAR
VAR
	Dummy					: U_64BIT_DATATYPE;
END_VAR

	Dummy._LWORD			:= In;
	Dummy._LWORD			:= SWAP_WORDS_OF_LWORD(Dummy._LWORD);
	
	IF	IsFinite(F_LREAL(dummy._LREAL)) THEN
		LWORD_TO_LREAL_EX 	:= dummy._LREAL;
	ELSE
		LWORD_TO_LREAL_EX	:= 0.0;
	END_IF

END_FUNCTION

// ---- POUs/_Miscellaneous/FbBaseExt.TcPOU
//Template for PlcOpen FB implementations with local path variable filled by attribute 'instance-path'
{attribute 'reflection'}
FUNCTION_BLOCK FbBaseExt EXTENDS FbBase
VAR_INPUT
END_VAR
VAR_IN_OUT
END_VAR
VAR_OUTPUT
    {attribute 'instance-path'}
    {attribute 'no_init'}
    Path  													: STRING;
END_VAR
VAR 
END_VAR
VAR
END_VAR

END_FUNCTION_BLOCK

// ---- POUs/_Miscellaneous/TEST_FB.TcPOU
//Should be called after new FBs to test signal flow and behavior of PlcOpen related variables 
FUNCTION_BLOCK Test_FB
VAR_OUTPUT CONSTANT
	NO_ERR 													:	INT := 0;
 	OK														:	INT := 1;
	ERR_BUSY 												:	INT := 2;
	ERR_DONE 												:	INT := 3;	
	ERR_ERR 												:	INT := 4;
	ERR_DONE_ERROR											:	INT := 5;
	ERR_NO_SIGNAL											:	INT := 6;
END_VAR             										
VAR_INPUT           										
	Reset													:	BOOL;	//The function block will be reset with a rising edge 
	Execute													:	BOOL;	//Link with Execute of the Fb to be tested
	Busy													:	BOOL;	//link with Busy Output of FB to be tested
	Error													:	BOOL;	//link with Error Output of FB to be tested
	Done													:	BOOL;	//link with Done Output of FB to be tested
END_VAR
VAR_OUTPUT
	ErrorId			:	INT := 0;	//Error identification 
END_VAR
VAR
	state			:	INT;
END_VAR

IF Reset
THEN
	state 													:= 0;
	ErrorId 												:= NO_ERR;
ELSE

	CASE state OF
	0:
		IF Execute
		THEN
			Errorid 										:= NO_ERR;
			IF Busy     									
			THEN        									
				state 										:= 10;
			ELSIF Error 									
			THEN        									
				state 										:= 20;
			ELSE        									
				state										:= state * -1;
				ErrorId 									:= ERR_BUSY;
			END_IF
		END_IF

	10:
		IF NOT Busy
		THEN
			IF Done
				AND Error
			THEN
				state										:= state * -1;
				ErrorId 									:= ERR_DONE_ERROR;
			ELSIF Done
			THEN
				IF Execute
				THEN
					state 									:= 11;
				ELSE      									
					state 									:= 12;
				END_IF
			ELSIF Error
			THEN
				IF Execute
				THEN
					state 									:= 21;
				ELSE      									
					state 									:= 22;
				END_IF
			ELSE
				state										:= state * -1;
				ErrorId 									:= ERR_NO_SIGNAL;
			END_IF
		END_IF

	11: (* Done muss wegsein wenn Execute nicht mehr da *)
		IF NOT Execute
		THEN
			IF NOT Done
			THEN
				state										:= 99;
			ELSE                							
				state										:= state * -1;
				ErrorId 									:= ERR_DONE;
			END_IF
		END_IF

	12: (* Done muss wegsein weil nur ein Zyklus *)
		IF NOT Done
		THEN
			state 											:= 99;
		ELSE
			state											:= state * -1;
			ErrorId 										:= ERR_DONE;
		END_IF


	20: (* Error Ohne Busy *)
		IF NOT Execute
		THEN
			IF Done
			THEN
				state										:= state * -1;
				ErrorId 									:= ERR_DONE;
			ELSIF Busy          							
			THEN                							
				state										:= state * -1;
				ErrorId 									:= ERR_BUSY;
			ELSE                	
				state										:= 99;
			END_IF
		END_IF

	21: (* Error muss wegsein wenn Execute nicht mehr da *)
		IF NOT Execute
		THEN
			IF NOT Error
			THEN
				state									:= 99;
			ELSE                						
				state									:= state * -1;
				ErrorId 								:= ERR_ERR;
			END_IF
		END_IF


	22: (* Error muss wegsein weil nur ein Zyklus *)
		IF NOT Error
		THEN
			state 										:= 99;
		ELSE                							
			state										:= state * -1;
			ErrorId 									:= ERR_DONE;
		END_IF              							
                            							
                            	
	99:                     	
		ErrorId											:= OK;
		state											:= 0;

	ELSE
		;
	END_CASE


END_IF

END_FUNCTION_BLOCK

// ---- POUs/Motion/TF50xx-NC/03_Utilities/AxStatemodel.TcPOU
{attribute 'no_check'}
//based on Statemodel instance
//IMPORTANT call this functionblock after AxAdmin !!!!
FUNCTION_BLOCK AxStatemodel EXTENDS Statemodel_Unit
VAR_INPUT 
	SafetyOK												:	BOOL := TRUE; //Drive safety card OK
	ENDisableInAborting										:	BOOL := FALSE; //Disable the axis directly in aborting instead of executing MC_Stop with given emergency dynamics  
	ENSoEReset												:	BOOL := TRUE; 
	ErrorActive												:	BOOL := FALSE; //Axis in error	
	EmergencyDec											:	LREAL := 0.0; //Emergency dec used in Aborting 
	EmergencyJerk											:	LREAL := 0.0; //Emergency jekr used in Aborting 
	rAxis													:	REFERENCE TO AXIS_REF := 0;
END_VAR
VAR_OUTPUT
END_VAR
VAR
	MC_Stop													: 	MC_Stop;
	MC_Reset												:	MC_Reset;
	SOE_Reset												:	FB_SoEReset;
	Mainstate												:	INT := 0;
	Ton_Seq													:	TON;
{attribute 'displaymode':='binary'}
	MemAbortingStep											:	BYTE; //Show online reasons for the aporting steps
END_VAR

	(* Axis UnitStateCtrl				 		V1.3		*)
	(*														*)
	(********************************************************)

(* check rAxis ************************************************)
IF NOT __ISVALIDREF(rAxis) 
THEN 
(*	ErrorText			:= 'Pointer pAxis invalid (0)'; *)
	RETURN;
END_IF

(* work local sub ****************************************)
	unit.name			:= CONCAT('Unit Axis ID: ', UDINT_TO_STRING(rAxis.NcToPlc.AxisId));

(* Call super ***************************************)
	SUPER^(); //Execute generic unit
		
(*********************************************************)

METHOD PROTECTED aborted : BOOL //Return value = TRUE if execution finsihed
VAR_INPUT
END_VAR
rAxis.PlcToNc.ControlDWord.0 						:= FALSE; (* Enable *)
rAxis.PlcToNc.ControlDWord.1 						:= FALSE; (* Enable_Positive *)
rAxis.PlcToNc.ControlDWord.2 						:= FALSE; (* Enable_Negative *)

MC_Stop(
	Axis			:= rAxis,
	Execute			:= 	MC_Stop.Execute 
						AND F_AxisControlLoopClosed(stateDWord := rAxis.NcToPlc.stateDWord) 
						AND rAxis.Status.PTPmode ,  (* Block new motion cmd *)
	Deceleration	:= ,
	Jerk			:= ,
	Options			:= ,
	Done			=> ,
	Busy			=> ,
	Active			=> ,
	CommandAborted	=> ,
	Error			=> ,
	ErrorID			=> );
	
Aborted												:= MC_Stop.Done OR MC_Stop.Error OR NOT F_AxisControlLoopClosed(stateDWord := rAxis.NcToPlc.stateDWord);
END_METHOD

METHOD PROTECTED aborting : BOOL //Return value = TRUE if execution finsihed
VAR_INPUT
END_VAR
CASE Mainstate OF
		0: (* Step 1 -> start stopping *)
			MemAbortingStep									:= 0;
			IF NOT rAxis.Status.PTPmode
				OR rAxis.Status.ProtectedMode
				OR rAxis.Status.MotionCommandsLocked
				OR NOT rAxis.Status.Operational
			THEN (* axis is slave-axis *)
				Mainstate									:= 99;
				MemAbortingStep.7							:= TRUE; 
			ELSIF ENDisableInAborting
			THEN
				rAxis.PlcToNc.ControlDWord.0 				:= FALSE; (* Enable *)
				rAxis.PlcToNc.ControlDWord.1 				:= FALSE; (* Enable_Positive *)
				rAxis.PlcToNc.ControlDWord.2 				:= FALSE; (* Enable_Negative *)
				MemAbortingStep.2							:= TRUE;
				Mainstate									:= 99;	
			ELSE
				IF NOT MC_Stop.busy      					
				THEN                        					
					MemAbortingStep.1						:= TRUE;
					Mainstate								:= 99;
				END_IF

				MC_Stop(
					Axis			:= rAxis,
					Execute			:= Mainstate = 99 ,
					Deceleration	:= EmergencyDec,(* NOT-HALT Parameter uebergeben *)
					Jerk			:= EmergencyJerk, (* NOT-HALT Parameter uebergeben *)
					Options			:= ,
					Done			=> ,
					Busy			=> ,
					Active			=> ,
					CommandAborted	=> ,
					Error			=> ,
					ErrorID			=> );
			END_IF

		99: (* Step 2 -> if stopped or safety signal = FALSE *) 
			MC_Stop(
				Axis			:= rAxis,
				Execute			:= ,
				Deceleration	:= ,
				Jerk			:= ,
				Options			:= ,
				Done			=> ,
				Busy			=> ,
				Active			=> ,
				CommandAborted	=> ,
				Error			=> ,
				ErrorID			=> );

			IF NOT F_AxisControlLoopClosed(stateDWord := rAxis.NcToPlc.stateDWord)
			THEN
				MemAbortingStep.4							:= TRUE;
				Unit.StateComplete();
				Aborting									:= TRUE;			
			ELSIF MC_Stop.Execute AND rAxis.Status.NotMoving AND (MC_Stop.Done OR MC_Stop.Error)	
			THEN                        					
				MemAbortingStep.3							:= TRUE;
				Unit.StateComplete();
				Aborting									:= TRUE;
			END_IF
		END_CASE
END_METHOD

METHOD PROTECTED clearing : BOOL //Return value = TRUE if execution finsihed
VAR_INPUT
END_VAR
CASE Mainstate OF
0:
	MC_Stop(
		Axis			:= rAxis,
		Execute			:= FALSE,
		Deceleration	:= , 
		Jerk			:= , 
		Options			:= , 
		Done			=> , 
		Busy			=> , 
		Active			=> , 
		CommandAborted	=> , 
		Error			=> , 
		ErrorID			=> );
		
	IF NOT MC_Stop.Busy
	THEN
		Mainstate									:= 99;
	END_IF
				
99:
	IF NOT rAxis.PlcToNc.ControlDWord.0 (* Enable is already active *)
		OR F_AxisControlLoopClosed(stateDWord := rAxis.NcToPlc.stateDWord)
		OR ErrorActive
	THEN
		Clearing									:= TRUE;
		Unit.StateComplete();
	END_IF
			
END_CASE
END_METHOD

METHOD PROTECTED completing : Bool //Return value = TRUE if execution finsihed
VAR_INPUT
END_VAR
(* Fehler ausloesen *)
IF UNit.InCompleting
	AND NOT F_AxisHasJob(stateDWord := rAxis.NcToPlc.stateDWord)
THEN
	Unit.StateComplete();
	Completing											:= TRUE;
ELSE
	Completing 											:= Executing();
END_IF
END_METHOD

METHOD PROTECTED executing : booL
VAR_INPUT
END_VAR
(* Set statemodel to error if axis is in error *********)
IF rAxis.NcToPlc.ErrorCode <> 0 OR ErrorActive 
THEN
	IF unit.optEnableFwdMachineErrorToMaster
	THEN
		Unit.SetMachineError();
	ELSE
		Unit.SetLocalError();
	END_IF
END_IF
	
Executing 												:= Unit.isStateActive(Unit.State);
END_METHOD

METHOD PROTECTED resetting : Bool //Return value = TRUE if execution finsihed
VAR_INPUT
END_VAR
		CASE Mainstate OF
		0:
			Ton_Seq(IN := FALSE);
			
			MC_Reset(
				Axis		:= rAxis,
				Execute		:= FALSE);
				
			SOE_Reset(
				Axis		:= rAxis,
				Execute		:= FALSE);

			IF SOE_Reset.Busy
				OR MC_Reset.Busy
			THEN
				;
			ELSIF SafetyOK
			THEN
				Mainstate									:= 10;
			ELSE            								
				Mainstate									:= 1;
			END_IF          	

		1: (* Wartezeit bis Safety OK *)
			Ton_Seq(IN := TRUE, PT := T#3S);
			IF SafetyOK	
			THEN
				Mainstate									:= 2;
			ELSIF Ton_Seq.Q 
			THEN (* Karten nicht resetbar .... *)
				Ton_Seq(IN := FALSE);
				Mainstate									:= 10;
			END_IF
			

		2: (* Wartezeit nach Safety Reset *)
			Ton_Seq(IN :=TRUE, PT := T#100MS);
			IF Ton_Seq.Q
			THEN
				Ton_Seq(IN := FALSE);
				Mainstate									:= 10;
			END_IF

		10: 
			SOE_Reset(
				Axis	:= rAxis,
				Execute	:= ENSoEReset AND(rAxis.Status.Error OR rAxis.Status.DriveDeviceError));

			Mainstate										:= 11;

		11:
			SOE_Reset(Axis	:= rAxis);
			IF NOT SOE_Reset.Busy THEN
				Mainstate			:= 20;
			END_IF

		20:
			MC_Reset(
				Axis	:= rAxis,
				Execute	:= NOT rAxis.Status.ProtectedMode OR rAxis.Status.Error);

			Mainstate										:= 21;

		21:
			MC_Reset( Axis	:= rAxis);
			IF NOT MC_Reset.Busy 
			THEN
				Mainstate									:= 99;
				Ton_Seq(IN := FALSE);
			END_IF

		99:
			Ton_Seq(IN := TRUE, PT := T#3S);
			MC_Reset(
				Axis	:= rAxis,
				Execute	:= FALSE);
				
			SOE_Reset(
				Axis	:= rAxis,
				Execute	:= FALSE);

			IF NOT MC_Reset.Busy
				AND NOT SOE_Reset.Busy
				AND(Ton_Seq.Q OR NOT ErrorActive AND NOT rAxis.Status.Error) 
			THEN
				Unit.StateComplete();
				Resetting									:= TRUE;
			END_IF
		END_CASE
END_METHOD

METHOD PROTECTED starting : Bool
VAR_INPUT
END_VAR
Unit.StateComplete();
Starting													:= Executing();
END_METHOD

METHOD PROTECTED stateChanged : BOOL 
VAR_INPUT
	mode											:	eMODE;
	state											:	eSTATE;
END_VAR
	MainState 										:= 0;
END_METHOD

METHOD PROTECTED stopped : Bool //Return value = TRUE if execution finsihed
VAR_INPUT
END_VAR
		MC_Stop(
			Axis			:= rAxis,
			Execute			:= FALSE,
			Deceleration	:= ,
			Jerk			:= ,
			Options			:= ,
			Done			=> ,
			Busy			=> ,
			Active			=> ,
			CommandAborted	=> ,
			Error			=> ,
			ErrorID			=> );
			
		Stopped													:= MC_Stop.Done OR MC_Stop.Error;
END_METHOD

METHOD PROTECTED stopping : BOOL //Return value = TRUE if execution finsihed
VAR_INPUT
END_VAR
		CASE Mainstate OF
		0:
			IF NOT MC_Stop.busy
			THEN
				Mainstate									:= 1;
			END_IF		

			MC_Stop(
				Axis			:= rAxis,
				Execute			:= 	Mainstate <> 0 
									AND NOT rAxis.Status.ProtectedMode 
									AND rAxis.Status.PTPmode,
				Deceleration	:= ,
				Jerk			:= ,
				Options			:= ,
				Done			=> ,
				Busy			=> ,
				Active			=> ,
				CommandAborted	=> ,
				Error			=> ,
				ErrorID		=> );

		1:
			MC_Stop(
				Axis			:= rAxis,
				Execute			:= 	MC_Stop.Execute 
									AND NOT rAxis.Status.NotMoving 
									AND rAxis.Status.ControlLoopClosed, (* Not Moving or not Operational *)
				Deceleration	:= ,
				Jerk			:= ,
				Options			:= ,
				Done			=> ,
				Busy			=> ,
				Active			=> ,
				CommandAborted	=> ,
				Error			=> ,
				ErrorID			=> );

			IF NOT MC_Stop.Execute AND NOT MC_Stop.Busy
			THEN
				Mainstate									:= 99;				
			END_IF
			
		99:
			Unit.StateComplete();
			Stopping										:= TRUE;
		END_CASE
END_METHOD

END_FUNCTION_BLOCK

// ---- POUs/Motion/TF50xx-NC/AxNcBaseExt.TcPOU
FUNCTION_BLOCK AxNcBaseExt EXTENDS AxNcBase 
VAR_OUTPUT CONSTANT
END_VAR
VAR_INPUT
	State													:	AxStatemodel;                                               
END_VAR                                             	
VAR_OUTPUT                                          	
END_VAR
VAR
END_VAR

	(* Axis 																*)
	(************************************************************************)

	
(********************************************************************************)
(* Call super 																	*)
(********************************************************************************)
	SUPER^();

(********************************************************************************)
(* Execute unit state model														*)
(********************************************************************************)
	State(
		Unit						:=  ,
		rAxis						:= THIS^,
		ENDisableInAborting			:= ,
		SafetyOK					:= ,//NOT Drive.SafetyError,
		ErrorActive					:= Event.ErrorId <> 0);

	//Execute aller Bausteine zuruecknehmen
	IF state.unit.InResetting 
		AND State.unit.RT_StateChanged
	THEN
		NoAction();
	END_IF

(********************************************************************************)

END_FUNCTION_BLOCK

// ---- POUs/Motion/TF5100-NCI/01_Main/NciItp.TcPOU
//Nci Interpolation group control - load,start,stop Nci programs as well start interpolated moves via Plc table (Tc2_PlcInterpolation library)
//based on Tc2_NCI, TcNcCfg.lib, Tc2_PlcInterpolation librarys
FUNCTION_BLOCK NciItp  EXTENDS FbBase
VAR_OUTPUT CONSTANT
	FNC_RESET												:	INT := 0; //Reset Nci group
	FNC_LOAD												:	INT := 1; //Load Nci program as txt/nc file
	FNC_START												:	INT := 2; //Start loaded Nci program
	FNC_STOP												:	INT := 3; //Stop loaded Nci programm
	FNC_FEED_TBL											:	INT := 4; //Feed table group - provided by Tc2_PlcInterpolation library
END_VAR                     								
VAR_INPUT                   								
	Fnc														:	INT (FNC_RESET..FNC_FEED_TBL):= FNC_RESET;
	Prg														:	T_MaxString := '';	//Program
	rTable													:	REFERENCE TO ST_NciFeedGroupTable := 0; //-> NciItpTableEntry
	rNCIRef													:	REFERENCE TO NCI_REF := 0;
	StartPrgAfterLoading									:	BOOL := FALSE; //Return value TRUE = Start Program direct after loading 
	LogFeederEntries										:	BOOL := FALSE; //Return value TRUE = Log tabel entries by Fnc FeedTbl
	WaitForChnDoneByEndOfTbl								:	BOOL := FALSE; //Fnc FeedTabl - TRUE = FB is busy as long as the prg is running if table contains entry "ST_NciEndOfTables"
END_VAR                     								
VAR_IN_OUT                  								
END_VAR                     								
VAR_OUTPUT                  								
	ErrorText												:	STRING(40);
END_VAR
VAR
(* cache **************************************************************************)
	MemFnc													:	INT := -1;
	MemResetAfterStop										:	BOOL;
                            								
(* timer *)                 								
                            	
(* trigger *)               	

(* MC-Function-block intances ******************************************************)
	ItpLoadProgEx											:	ItpLoadProgEx;
	ItpStartStopEx											:	ItpStartStopEx;
	NciFeedTable											:	FB_NciFeedTable;
	ItpResetEx2												:	ItpResetEx2 := (tTimeOut	:= DEFAULT_ADS_TIMEOUT);

END_VAR

	(* NCI Program control																*)
	(************************************************************************************)

(* Execute ***************************************************************************************)
	rtExecute(CLK := Execute );
	IF rtExecute.Q
		AND MemFnc < 0
	THEN
		MemFnc 												:= Fnc;
		Busy												:= TRUE;
		Done												:= FALSE;
		Error												:= FALSE;
		ErrorID												:= 0;
		ErrorText											:= '';
	END_IF

(* Call Method ***********************************************************************************)
	CASE MemFnc OF
	FNC_RESET							:
		Reset(Execute:= Execute);
	FNC_LOAD							:
		LoadPrg(Execute:= Execute, Prg:= Prg);
	FNC_START							:
		StartPrg(Execute:= Execute);
	FNC_STOP							:
		StopPrg(Execute:= Execute);
	FNC_FEED_TBL						:
		FeedTbl(Execute:= Execute );
	-1:
		IF NOT Execute
		THEN
			Busy											:= FALSE;
			Done											:= FALSE;
			Error											:= FALSE;
			ErrorID											:= 0;
			ErrorText										:= '';
		END_IF                              				
	ELSE                                    				
		Busy												:= FALSE;
		Done												:= FALSE;
		Error												:= Execute;
		ErrorID												:= E_AdsErr.DEVICE_INVALIDPARM;
		ErrorText											:= CONCAT('invalid parameter value(s) Fnc no: ' , INT_TO_STRING(MemFnc));
	END_CASE


(**************************************************************************************************)

METHOD PUBLIC feedTbl : BOOL //Return value = TRUE if busy
//required parameter
//rNCIRef
//rTable
VAR_INPUT
	Execute													:	BOOL := FALSE;
END_VAR
	MemFnc													:= FNC_FEED_TBL;
	THIS^.Execute											:= Execute;
	
IF NOT __ISVALIDREF(rNCIRef) 
THEN
	Busy													:= NOT Error;
	Error													:= TRUE;
	ErrorId													:= E_AdsErr.DEVICE_INVALIDPARM;
	Done													:= FALSE;
	ErrorText												:= 'Reference rNCIRef invalid (0)';
	MemFnc													:= SEL(Execute , -1 ,MemFnc); 
	RETURN;
ELSIF NOT __ISVALIDREF(rTable) 
THEN
	Busy													:= NOT Error;
	Error													:= TRUE;
	ErrorId													:= E_AdsErr.DEVICE_INVALIDPARM;
	Done													:= FALSE;
	ErrorText												:= 'Reference rTable invalid (0)';
	MemFnc													:= SEL(Execute , -1 ,MemFnc);
	RETURN;
END_IF

	IF Execute
	THEN
		Error												:=	FALSE;
		ErrorId												:= 0;
		NciFeedTable.bExecute 								:= TRUE;
	ELSIF NOT NciFeedTable.bFeedBusy
		AND(
		NOT NciFeedTable.bExecChannelDoneCheck
		OR NciFeedTable.bChannelDone)
	THEN
		Error												:=	FALSE;
		ErrorId												:= 0;
		NciFeedTable.bExecute 								:= FALSE;
	END_IF

	NciFeedTable(
		bExecute			:= ,
		bReset				:= FALSE,
		bLogFeederEntries	:= LogFeederEntries,
		stFeedGroupTable	:= rTable,
		stNciToPlc			:= rNCIRef.NciToPlc,
		bFeedingDone		=> 	,
		bChannelDone		=> ,
		bFeedBusy			=> ,
		bResetBusy			=> ,
		bError				=> ,
		nErrorId			=> );

	IF WaitForChnDoneByEndOfTbl
	THEN
		Busy 												:= NciFeedTable.bFeedBusy
																OR
																NciFeedTable.bFeedingDone
																AND NciFeedTable.bExecChannelDoneCheck
																AND NOT NciFeedTable.bChannelDone;
                            								
		Done												:= NciFeedTable.bChannelDone
																OR
																NciFeedTable.bFeedingDone
																AND NOT NciFeedTable.bExecChannelDoneCheck;
                            								
	ELSE                    								
		Busy												:= NciFeedTable.bFeedBusy;
		Done												:= NciFeedTable.bFeedingDone;
	END_IF

	IF NOT Busy
	THEN
		IF NciFeedTable.bExecute
		THEN
			Error											:=	NciFeedTable.bError;
			ErrorId											:= NciFeedTable.nErrorId;
			ErrorText										:= SEL(Error , '' ,  CONCAT('Error NciFeedTable id: ',  UDINT_TO_STRING(Errorid)));
		END_IF                          					
		IF NOT Execute                  					
		THEN                            					
			MemFnc											:= -1 ;
			NciFeedTable(bExecute 							:= FALSE, stNciToPlc:= rNCIRef.NciToPlc, stFeedGroupTable:= rTable  );
		END_IF                          	
	END_IF                              	
                                        	
	FeedTbl													:= Busy;
END_METHOD

METHOD PUBLIC loadPrg : BOOL //Return value = TRUE if busy
//required parameter
//rNCIRef
VAR_INPUT
	Execute													:	BOOL;
	Prg														:	T_MaxString := ''; //if Prg = '' then INPUT THIS^.Prg used
END_VAR
	MemFnc													:= FNC_LOAD;
	THIS^.Execute											:= Execute;
	
IF NOT __ISVALIDREF(rNCIRef) THEN
	Busy													:= NOT Error;
	Error													:= TRUE;
	ErrorId													:= E_AdsErr.DEVICE_INVALIDPARM;
	Done													:= FALSE;
	ErrorText												:= 'Reference rNCIRef invalid (0)';
	MemFnc													:= SEL(Execute , -1 ,MemFnc);
	RETURN;
END_IF
	
	IF Execute AND NOT ItpLoadProgEx.bExecute
	THEN
		IF LEN(Prg) > 0
		THEN
			ItpLoadProgEx.sPrg								:= Prg;
		ELSE                    							
			ItpLoadProgEx.sPrg								:= THIS^.Prg;	
		END_IF
	END_IF	
	
	IF Execute
	THEN
		Error												:=	FALSE;
		ErrorId												:= 0;
		ItpLoadProgEx.bExecute 								:= TRUE;
	ELSIF NOT ItpLoadProgEx.bBusy       					
		AND(                            					
		NOT ItpStartStopEx.bBusy        					
		OR NOT StartPrgAfterLoading)    					
	THEN                                					
		Error												:=	FALSE;
		ErrorId												:= 0;
		ItpLoadProgEx.bExecute 								:= FALSE;
		IF StartPrgAfterLoading             				
		THEN                                				
			ItpStartStopEx.bStart 							:= FALSE;
		END_IF
	END_IF
	
	ItpLoadProgEx(
		bExecute	:= ,
		sPrg		:= ,
		nLength		:= INT_TO_UDINT(LEN(Prg)),
		tTimeOut	:= ,
		sNciToPlc	:= rNCIRef.NciToPlc,
		bBusy		=> ,
		bErr		=> ,
		nErrId		=> );

	IF StartPrgAfterLoading
		OR ItpStartStopEx.bBusy
	THEN
		ItpStartStopEx(
			bStart		:= ItpLoadProgEx.bExecute
							AND NOT ItpLoadProgEx.bErr
							AND NOT ItpLoadProgEx.bBusy,
			bStop		:= FALSE,
			tTimeOut	:=  ,
			sNciToPlc	:= rNCIRef.NciToPlc,
			bBusy		=> ,
			bErr		=> ,
			nErrId		=> );
	END_IF


	Busy													:= ItpStartStopEx.bBusy OR ItpLoadProgEx.bBusy;
                                        					
